LIN {X 0,Y 333.716,Z 810.919,A -85,B 0,C 180,E1 -14697.808,E2 -14697.808} C_VEL
LIN {X 0,Y 333.692,Z 810.92,A -85,B 0,C 180,E1 -14700.36,E2 -14700.36} C_VEL
LIN {X 0,Y 333.667,Z 810.922,A -85,B 0,C 180,E1 -14704.656,E2 -14704.656} C_VEL
LIN {X 0,Y 333.648,Z 810.925,A -85,B 0,C 180,E1 -14707.648,E2 -14707.648} C_VEL
LIN {X 0,Y 333.69,Z 810.919,A -85,B 0,C 180,E1 -14710.757,E2 -14710.757} C_VEL
LIN {X 0,Y 333.72,Z 810.918,A -85,B 0,C 180,E1 -14714.272,E2 -14714.272} C_VEL
LIN {X 0,Y 333.695,Z 810.911,A -85,B 0,C 180,E1 -14717.627,E2 -14717.627} C_VEL
LIN {X 0,Y 333.676,Z 810.914,A -85,B 0,C 180,E1 -14721.193,E2 -14721.193} C_VEL
LIN {X 0,Y 333.644,Z 810.921,A -85,B 0,C 180,E1 -14722.65,E2 -14722.65} C_VEL
LIN {X 0,Y 332.983,Z 811.005,A -85,B 0,C 180,E1 -14723.657,E2 -14723.657} C_VEL
LIN {X 0,Y 330.131,Z 811.362,A -85,B 0,C 180,E1 -14725.297,E2 -14725.297} C_VEL
LIN {X 0,Y 327.705,Z 811.662,A -85,B 0,C 180,E1 -14726.625,E2 -14726.625} C_VEL
LIN {X 0,Y 326.655,Z 811.793,A -85,B 0,C 180,E1 -14727.654,E2 -14727.654} C_VEL
LIN {X 0,Y 326.565,Z 811.801,A -85,B 0,C 180,E1 -14728.002,E2 -14728.002} C_VEL
LIN {X 0,Y 326.643,Z 811.794,A -85,B 0,C 180,E1 -14731.748,E2 -14731.748} C_VEL
LIN {X 0,Y 326.674,Z 811.789,A -85,B 0,C 180,E1 -14734.626,E2 -14734.626} C_VEL
LIN {X 0,Y 326.633,Z 811.797,A -85,B 0,C 180,E1 -14738.544,E2 -14738.544} C_VEL
LIN {X 0,Y 326.729,Z 811.788,A -85,B 0,C 180,E1 -14741.176,E2 -14741.176} C_VEL
LIN {X 0,Y 326.747,Z 811.778,A -85,B 0,C 180,E1 -14745.432,E2 -14745.432} C_VEL
LIN {X 0,Y 326.758,Z 811.784,A -85,B 0,C 180,E1 -14748.838,E2 -14748.838} C_VEL
LIN {X 0,Y 326.949,Z 811.757,A -85,B 0,C 180,E1 -14752.59,E2 -14752.59} C_VEL
LIN {X 0,Y 326.76,Z 811.787,A -85,B 0,C 180,E1 -14755.065,E2 -14755.065} C_VEL
LIN {X 0,Y 327.03,Z 811.746,A -85,B 0,C 180,E1 -14757.537,E2 -14757.537} C_VEL
LIN {X 0,Y 327.181,Z 811.733,A -85,B 0,C 180,E1 -14760,E2 -14760} C_VEL
LIN {X 0,Y 327.029,Z 811.75,A -85,B 0,C 180,E1 -14762.463,E2 -14762.463} C_VEL
LIN {X 0,Y 326.945,Z 811.758,A -85,B 0,C 180,E1 -14766.17,E2 -14766.17} C_VEL
LIN {X 0,Y 326.898,Z 811.762,A -85,B 0,C 180,E1 -14768.655,E2 -14768.655} C_VEL
LIN {X 0,Y 326.721,Z 811.78,A -85,B 0,C 180,E1 -14772.422,E2 -14772.422} C_VEL
LIN {X 0,Y 326.738,Z 811.784,A -85,B 0,C 180,E1 -14774.958,E2 -14774.958} C_VEL
LIN {X 0,Y 326.717,Z 811.788,A -85,B 0,C 180,E1 -14778.839,E2 -14778.839} C_VEL
LIN {X 0,Y 326.582,Z 811.804,A -85,B 0,C 180,E1 -14782.79,E2 -14782.79} C_VEL
LIN {X 0,Y 326.619,Z 811.798,A -85,B 0,C 180,E1 -14785.49,E2 -14785.49} C_VEL
LIN {X 0,Y 326.601,Z 811.803,A -85,B 0,C 180,E1 -14789.665,E2 -14789.665} C_VEL
LIN {X 0,Y 326.603,Z 811.8,A -85,B 0,C 180,E1 -14792.947,E2 -14792.947} C_VEL
LIN {X 0,Y 326.596,Z 811.803,A -85,B 0,C 180,E1 -14795.522,E2 -14795.522} C_VEL
LIN {X 0,Y 326.573,Z 811.807,A -85,B 0,C 180,E1 -14799.223,E2 -14799.223} C_VEL
LIN {X 0,Y 326.595,Z 811.905,A -85,B 0,C 180,E1 -14801.33,E2 -14801.33} C_VEL
LIN {X 0,Y 327.886,Z 817.95,A -85,B 0,C 180,E1 -14804.156,E2 -14804.156} C_VEL
LIN {X 0,Y 329.434,Z 825.489,A -85,B 0,C 180,E1 -14807.477,E2 -14807.477} C_VEL
LIN {X 0,Y 331.048,Z 834.395,A -85,B 0,C 180,E1 -14811.14,E2 -14811.14} C_VEL
LIN {X 0,Y 331.312,Z 837.705,A -85,B 0,C 180,E1 -14812.424,E2 -14812.424} C_VEL
LIN {X 0,Y 329.861,Z 848.572,A -85,B 0,C 180,E1 -14816.364,E2 -14816.364} C_VEL
LIN {X 0,Y 328.321,Z 861.677,A -85,B 0,C 180,E1 -14821.019,E2 -14821.019} C_VEL
LIN {X 0,Y 327.361,Z 871.737,A -85,B 0,C 180,E1 -14824.575,E2 -14824.575} C_VEL
LIN {X 0,Y 326.643,Z 880.438,A -85,B 0,C 180,E1 -14827.625,E2 -14827.625} C_VEL
LIN {X 0,Y 328.711,Z 894.714,A -85,B 0,C 180,E1 -14828.278,E2 -14828.278} C_VEL
LIN {X 0,Y 329.806,Z 906.751,A -85,B 0,C 180,E1 -14829.017,E2 -14829.017} C_VEL
LIN {X 0,Y 330.337,Z 918.761,A -85,B 0,C 180,E1 -14829.954,E2 -14829.954} C_VEL
LIN {X 0,Y 330.378,Z 930.265,A -85,B 0,C 180,E1 -14831.073,E2 -14831.073} C_VEL
LIN {X 0,Y 330.455,Z 937.231,A -85,B 0,C 180,E1 -14831.881,E2 -14831.881} C_VEL
LIN {X 0,Y 329.062,Z 947.55,A -85,B 0,C 180,E1 -14833.245,E2 -14833.245} C_VEL
LIN {X 0,Y 327.748,Z 957.445,A -85,B 0,C 180,E1 -14834.881,E2 -14834.881} C_VEL
LIN {X 0,Y 326.998,Z 964.642,A -85,B 0,C 180,E1 -14836.327,E2 -14836.327} C_VEL
LIN {X 0,Y 326.251,Z 972.29,A -85,B 0,C 180,E1 -14838.194,E2 -14838.194} C_VEL
LIN {X 0,Y 325.834,Z 978.472,A -85,B 0,C 180,E1 -14840.066,E2 -14840.066} C_VEL
LIN {X 0,Y 325.696,Z 983.394,A -85,B 0,C 180,E1 -14841.939,E2 -14841.939} C_VEL
LIN {X 0,Y 325.738,Z 987.186,A -85,B 0,C 180,E1 -14843.809,E2 -14843.809} C_VEL
LIN {X 0,Y 325.892,Z 989.16,A -85,B 0,C 180,E1 -14845.054,E2 -14845.054} C_VEL
LIN {X 0,Y 326.004,Z 990.64,A -85,B 0,C 180,E1 -14846.294,E2 -14846.294} C_VEL
LIN {X 0,Y 326.056,Z 991.691,A -85,B 0,C 180,E1 -14847.532,E2 -14847.532} C_VEL
LIN {X 0,Y 326.14,Z 992.338,A -85,B 0,C 180,E1 -14848.767,E2 -14848.767} C_VEL
LIN {X 0,Y 326.213,Z 992.572,A -85,B 0,C 180,E1 -14850.002,E2 -14850.002} C_VEL
LIN {X 0,Y 326.141,Z 992.332,A -85,B 0,C 180,E1 -14851.237,E2 -14851.237} C_VEL
LIN {X 0,Y 326.057,Z 991.679,A -85,B 0,C 180,E1 -14852.473,E2 -14852.473} C_VEL
LIN {X 0,Y 326.005,Z 990.623,A -85,B 0,C 180,E1 -14853.71,E2 -14853.71} C_VEL
LIN {X 0,Y 325.893,Z 989.136,A -85,B 0,C 180,E1 -14854.951,E2 -14854.951} C_VEL
LIN {X 0,Y 325.738,Z 985.606,A -85,B 0,C 180,E1 -14857.03,E2 -14857.03} C_VEL
LIN {X 0,Y 325.757,Z 980.196,A -85,B 0,C 180,E1 -14859.314,E2 -14859.314} C_VEL
LIN {X 0,Y 326.028,Z 974.442,A -85,B 0,C 180,E1 -14861.189,E2 -14861.189} C_VEL
LIN {X 0,Y 326.71,Z 967.329,A -85,B 0,C 180,E1 -14863.056,E2 -14863.056} C_VEL
LIN {X 0,Y 327.555,Z 960.109,A -85,B 0,C 180,E1 -14864.604,E2 -14864.604} C_VEL
LIN {X 0,Y 329.351,Z 946.504,A -85,B 0,C 180,E1 -14867.064,E2 -14867.064} C_VEL
LIN {X 0,Y 330.884,Z 936.373,A -85,B 0,C 180,E1 -14868.58,E2 -14868.58} C_VEL
LIN {X 0,Y 331.378,Z 923.905,A -85,B 0,C 180,E1 -14870.201,E2 -14870.201} C_VEL
LIN {X 0,Y 331.81,Z 912.737,A -85,B 0,C 180,E1 -14871.432,E2 -14871.432} C_VEL
LIN {X 0,Y 331.901,Z 904.635,A -85,B 0,C 180,E1 -14872.243,E2 -14872.243} C_VEL
LIN {X 0,Y 330.655,Z 891.44,A -85,B 0,C 180,E1 -14873.499,E2 -14873.499} C_VEL
LIN {X 0,Y 328.27,Z 877.306,A -85,B 0,C 180,E1 -14874.788,E2 -14874.788} C_VEL
LIN {X 0,Y 327.341,Z 873.127,A -85,B 0,C 180,E1 -14875.176,E2 -14875.176} C_VEL
LIN {X 0,Y 327.288,Z 872.165,A -85,B 0,C 180,E1 -14875.266,E2 -14875.266} C_VEL
LIN {X 0,Y 328.289,Z 861.638,A -85,B 0,C 180,E1 -14878.985,E2 -14878.985} C_VEL
LIN {X 0,Y 329.588,Z 850.492,A -85,B 0,C 180,E1 -14882.941,E2 -14882.941} C_VEL
LIN {X 0,Y 331.19,Z 838.637,A -85,B 0,C 180,E1 -14887.215,E2 -14887.215} C_VEL
LIN {X 0,Y 331.22,Z 835.828,A -85,B 0,C 180,E1 -14888.271,E2 -14888.271} C_VEL
LIN {X 0,Y 329.746,Z 827.239,A -85,B 0,C 180,E1 -14891.758,E2 -14891.758} C_VEL
LIN {X 0,Y 327.846,Z 817.89,A -85,B 0,C 180,E1 -14895.837,E2 -14895.837} C_VEL
LIN {X 0,Y 326.561,Z 811.81,A -85,B 0,C 180,E1 -14898.772,E2 -14898.772} C_VEL
LIN {X 0,Y 326.629,Z 811.798,A -85,B 0,C 180,E1 -14902.953,E2 -14902.953} C_VEL
LIN {X 0,Y 326.611,Z 811.799,A -85,B 0,C 180,E1 -14905.981,E2 -14905.981} C_VEL
LIN {X 0,Y 326.616,Z 811.799,A -85,B 0,C 180,E1 -14909.399,E2 -14909.399} C_VEL
LIN {X 0,Y 326.6,Z 811.803,A -85,B 0,C 180,E1 -14913.135,E2 -14913.135} C_VEL
LIN {X 0,Y 326.614,Z 811.858,A -85,B 0,C 180,E1 -14914.424,E2 -14914.424} C_VEL
LIN {X 0,Y 326.863,Z 813.01,A -85,B 0,C 180,E1 -14914.566,E2 -14914.566} C_VEL
LIN {X 0,Y 327.872,Z 815.002,A -85,B 0,C 180,E1 -14914.913,E2 -14914.913} C_VEL
LIN {X 0,Y 329.004,Z 816.271,A -85,B 0,C 180,E1 -14915.215,E2 -14915.215} C_VEL
LIN {X 0,Y 331.968,Z 822.323,A -85,B 0,C 180,E1 -14916.281,E2 -14916.281} C_VEL
LIN {X 0,Y 335.858,Z 830.631,A -85,B 0,C 180,E1 -14917.76,E2 -14917.76} C_VEL
LIN {X 0,Y 339.022,Z 840.104,A -85,B 0,C 180,E1 -14919.365,E2 -14919.365} C_VEL
LIN {X 0,Y 339.722,Z 843.27,A -85,B 0,C 180,E1 -14919.896,E2 -14919.896} C_VEL
LIN {X 0,Y 338.28,Z 853.109,A -85,B 0,C 180,E1 -14921.215,E2 -14921.215} C_VEL
LIN {X 0,Y 336.922,Z 860.61,A -85,B 0,C 180,E1 -14922.394,E2 -14922.394} C_VEL
LIN {X 0,Y 335.4,Z 868.603,A -85,B 0,C 180,E1 -14923.88,E2 -14923.88} C_VEL
LIN {X 0,Y 333.761,Z 876.022,A -85,B 0,C 180,E1 -14925.614,E2 -14925.614} C_VEL
LIN {X 0,Y 332.03,Z 883.463,A -85,B 0,C 180,E1 -14927.78,E2 -14927.78} C_VEL
LIN {X 0,Y 330.34,Z 889.554,A -85,B 0,C 180,E1 -14930.201,E2 -14930.201} C_VEL
LIN {X 0,Y 329.629,Z 891.806,A -85,B 0,C 180,E1 -14931.417,E2 -14931.417} C_VEL
LIN {X 0,Y 328.897,Z 893.676,A -85,B 0,C 180,E1 -14932.634,E2 -14932.634} C_VEL
LIN {X 0,Y 328.111,Z 896.009,A -85,B 0,C 180,E1 -14935.085,E2 -14935.085} C_VEL
LIN {X 0,Y 327.478,Z 896.771,A -85,B 0,C 180,E1 -14937.54,E2 -14937.54} C_VEL
LIN {X 0,Y 327.203,Z 896.509,A -85,B 0,C 180,E1 -14938.769,E2 -14938.769} C_VEL
LIN {X 0,Y 326.915,Z 895.854,A -85,B 0,C 180,E1 -14940,E2 -14940} C_VEL
LIN {X 0,Y 326.782,Z 893.268,A -85,B 0,C 180,E1 -14942.465,E2 -14942.465} C_VEL
LIN {X 0,Y 326.755,Z 890.202,A -85,B 0,C 180,E1 -14944.317,E2 -14944.317} C_VEL
LIN {X 0,Y 327.16,Z 886.056,A -85,B 0,C 180,E1 -14946.166,E2 -14946.166} C_VEL
LIN {X 0,Y 327.526,Z 880.773,A -85,B 0,C 180,E1 -14948.018,E2 -14948.018} C_VEL
LIN {X 0,Y 327.848,Z 875.453,A -85,B 0,C 180,E1 -14949.559,E2 -14949.559} C_VEL
LIN {X 0,Y 328.493,Z 867.671,A -85,B 0,C 180,E1 -14951.414,E2 -14951.414} C_VEL
LIN {X 0,Y 329.086,Z 859.694,A -85,B 0,C 180,E1 -14952.958,E2 -14952.958} C_VEL
LIN {X 0,Y 329.713,Z 851.26,A -85,B 0,C 180,E1 -14954.347,E2 -14954.347} C_VEL
LIN {X 0,Y 330.285,Z 843.596,A -85,B 0,C 180,E1 -14955.425,E2 -14955.425} C_VEL
LIN {X 0,Y 331.05,Z 833.535,A -85,B 0,C 180,E1 -14956.638,E2 -14956.638} C_VEL
LIN {X 0,Y 331.244,Z 830.494,A -85,B 0,C 180,E1 -14956.954,E2 -14956.954} C_VEL
LIN {X 0,Y 328.32,Z 818.286,A -85,B 0,C 180,E1 -14958.217,E2 -14958.217} C_VEL
LIN {X 0,Y 326.633,Z 811.795,A -85,B 0,C 180,E1 -14958.806,E2 -14958.806} C_VEL
LIN {X 0,Y 326.59,Z 811.797,A -85,B 0,C 180,E1 -14962.79,E2 -14962.79} C_VEL
LIN {X 0,Y 326.601,Z 811.792,A -85,B 0,C 180,E1 -14966.865,E2 -14966.865} C_VEL
LIN {X 0,Y 326.58,Z 811.8,A -85,B 0,C 180,E1 -14971.097,E2 -14971.097} C_VEL
LIN {X 0,Y 326.613,Z 811.796,A -85,B 0,C 180,E1 -14974.019,E2 -14974.019} C_VEL
LIN {X 0,Y 326.628,Z 811.791,A -85,B 0,C 180,E1 -14977.236,E2 -14977.236} C_VEL
LIN {X 0,Y 326.551,Z 811.804,A -85,B 0,C 180,E1 -14981.124,E2 -14981.124} C_VEL
LIN {X 0,Y 326.568,Z 811.802,A -85,B 0,C 180,E1 -14983.525,E2 -14983.525} C_VEL
LIN {X 0,Y 326.581,Z 811.801,A -85,B 0,C 180,E1 -14987.028,E2 -14987.028} C_VEL
LIN {X 0,Y 326.593,Z 811.802,A -85,B 0,C 180,E1 -14990.777,E2 -14990.777} C_VEL
LIN {X 0,Y 326.619,Z 811.801,A -85,B 0,C 180,E1 -14994.479,E2 -14994.479} C_VEL
LIN {X 0,Y 326.615,Z 811.797,A -85,B 0,C 180,E1 -14997.454,E2 -14997.454} C_VEL
LIN {X 0,Y 326.654,Z 811.79,A -85,B 0,C 180,E1 -15000.338,E2 -15000.338} C_VEL
LIN {X 0,Y 326.696,Z 811.783,A -85,B 0,C 180,E1 -15004.515,E2 -15004.515} C_VEL
LIN {X 0,Y 326.65,Z 811.826,A -85,B 0,C 180,E1 -15008.544,E2 -15008.544} C_VEL
LIN {X 0,Y 330.897,Z 823.77,A -85,B 0,C 180,E1 -15009.727,E2 -15009.727} C_VEL
LIN {X 0,Y 334.128,Z 834.117,A -85,B 0,C 180,E1 -15010.94,E2 -15010.94} C_VEL
LIN {X 0,Y 334.837,Z 836.764,A -85,B 0,C 180,E1 -15011.276,E2 -15011.276} C_VEL
LIN {X 0,Y 333.841,Z 847.507,A -85,B 0,C 180,E1 -15012.541,E2 -15012.541} C_VEL
LIN {X 0,Y 332.661,Z 857.844,A -85,B 0,C 180,E1 -15014.057,E2 -15014.057} C_VEL
LIN {X 0,Y 331.579,Z 866.207,A -85,B 0,C 180,E1 -15015.577,E2 -15015.577} C_VEL
LIN {X 0,Y 330.347,Z 874.325,A -85,B 0,C 180,E1 -15017.403,E2 -15017.403} C_VEL
LIN {X 0,Y 329.595,Z 879.852,A -85,B 0,C 180,E1 -15018.934,E2 -15018.934} C_VEL
LIN {X 0,Y 328.829,Z 885.233,A -85,B 0,C 180,E1 -15020.774,E2 -15020.774} C_VEL
LIN {X 0,Y 327.901,Z 889.497,A -85,B 0,C 180,E1 -15022.609,E2 -15022.609} C_VEL
LIN {X 0,Y 327.572,Z 891.723,A -85,B 0,C 180,E1 -15023.84,E2 -15023.84} C_VEL
LIN {X 0,Y 327.275,Z 893.539,A -85,B 0,C 180,E1 -15025.07,E2 -15025.07} C_VEL
LIN {X 0,Y 327.271,Z 894.875,A -85,B 0,C 180,E1 -15026.304,E2 -15026.304} C_VEL
LIN {X 0,Y 326.973,Z 896.453,A -85,B 0,C 180,E1 -15028.766,E2 -15028.766} C_VEL
LIN {X 0,Y 326.926,Z 896.684,A -85,B 0,C 180,E1 -15029.998,E2 -15029.998} C_VEL
LIN {X 0,Y 327.106,Z 895.92,A -85,B 0,C 180,E1 -15032.461,E2 -15032.461} C_VEL
LIN {X 0,Y 327.23,Z 894.981,A -85,B 0,C 180,E1 -15033.692,E2 -15033.692} C_VEL
LIN {X 0,Y 327.263,Z 893.685,A -85,B 0,C 180,E1 -15034.926,E2 -15034.926} C_VEL
LIN {X 0,Y 327.73,Z 890.88,A -85,B 0,C 180,E1 -15036.771,E2 -15036.771} C_VEL
LIN {X 0,Y 328.576,Z 887.039,A -85,B 0,C 180,E1 -15038.609,E2 -15038.609} C_VEL
LIN {X 0,Y 329.297,Z 882.586,A -85,B 0,C 180,E1 -15040.287,E2 -15040.287} C_VEL
LIN {X 0,Y 330.101,Z 875.962,A -85,B 0,C 180,E1 -15042.29,E2 -15042.29} C_VEL
LIN {X 0,Y 331.295,Z 868.186,A -85,B 0,C 180,E1 -15044.118,E2 -15044.118} C_VEL
LIN {X 0,Y 332.365,Z 860.257,A -85,B 0,C 180,E1 -15045.638,E2 -15045.638} C_VEL
LIN {X 0,Y 333.544,Z 850.564,A -85,B 0,C 180,E1 -15047.154,E2 -15047.154} C_VEL
LIN {X 0,Y 334.7,Z 839.753,A -85,B 0,C 180,E1 -15048.501,E2 -15048.501} C_VEL
LIN {X 0,Y 334.99,Z 837.259,A -85,B 0,C 180,E1 -15048.765,E2 -15048.765} C_VEL
LIN {X 0,Y 331.653,Z 825.781,A -85,B 0,C 180,E1 -15050.157,E2 -15050.157} C_VEL
LIN {X 0,Y 327.543,Z 814.401,A -85,B 0,C 180,E1 -15051.331,E2 -15051.331} C_VEL
LIN {X 0,Y 326.666,Z 811.794,A -85,B 0,C 180,E1 -15051.573,E2 -15051.573} C_VEL
LIN {X 0,Y 326.686,Z 811.793,A -85,B 0,C 180,E1 -15055.481,E2 -15055.481} C_VEL
LIN {X 0,Y 326.655,Z 811.797,A -85,B 0,C 180,E1 -15059.657,E2 -15059.657} C_VEL
LIN {X 0,Y 326.601,Z 811.805,A -85,B 0,C 180,E1 -15064.017,E2 -15064.017} C_VEL
LIN {X 0,Y 326.622,Z 811.799,A -85,B 0,C 180,E1 -15067.237,E2 -15067.237} C_VEL
LIN {X 0,Y 326.627,Z 811.802,A -85,B 0,C 180,E1 -15070.2,E2 -15070.2} C_VEL
LIN {X 0,Y 326.649,Z 811.795,A -85,B 0,C 180,E1 -15073.507,E2 -15073.507} C_VEL
LIN {X 0,Y 326.64,Z 811.791,A -85,B 0,C 180,E1 -15077.012,E2 -15077.012} C_VEL
LIN {X 0,Y 326.636,Z 811.793,A -85,B 0,C 180,E1 -15080.763,E2 -15080.763} C_VEL
LIN {X 0,Y 326.602,Z 811.801,A -85,B 0,C 180,E1 -15084.479,E2 -15084.479} C_VEL
LIN {X 0,Y 326.565,Z 811.801,A -85,B 0,C 180,E1 -15088.002,E2 -15088.002} C_VEL
LIN {X 0,Y 325.885,Z 811.888,A -85,B 0,C 180,E1 -15089.033,E2 -15089.033} C_VEL
LIN {X 0,Y 323.038,Z 812.242,A -85,B 0,C 180,E1 -15090.711,E2 -15090.711} C_VEL
LIN {X 0,Y 320.653,Z 812.541,A -85,B 0,C 180,E1 -15092.07,E2 -15092.07} C_VEL
LIN {X 0,Y 319.658,Z 812.664,A -85,B 0,C 180,E1 -15093.122,E2 -15093.122} C_VEL
LIN {X 0,Y 319.592,Z 812.669,A -85,B 0,C 180,E1 -15093.478,E2 -15093.478} C_VEL
LIN {X 0,Y 319.594,Z 812.673,A -85,B 0,C 180,E1 -15097.45,E2 -15097.45} C_VEL
LIN {X 0,Y 319.674,Z 812.665,A -85,B 0,C 180,E1 -15100.961,E2 -15100.961} C_VEL
LIN {X 0,Y 319.715,Z 812.653,A -85,B 0,C 180,E1 -15105.275,E2 -15105.275} C_VEL
LIN {X 0,Y 319.743,Z 812.65,A -85,B 0,C 180,E1 -15109.872,E2 -15109.872} C_VEL
LIN {X 0,Y 319.908,Z 812.634,A -85,B 0,C 180,E1 -15112.426,E2 -15112.426} C_VEL
LIN {X 0,Y 319.729,Z 812.662,A -85,B 0,C 180,E1 -15114.956,E2 -15114.956} C_VEL
LIN {X 0,Y 319.974,Z 812.625,A -85,B 0,C 180,E1 -15117.482,E2 -15117.482} C_VEL
LIN {X 0,Y 320.133,Z 812.611,A -85,B 0,C 180,E1 -15120,E2 -15120} C_VEL
LIN {X 0,Y 319.972,Z 812.629,A -85,B 0,C 180,E1 -15122.518,E2 -15122.518} C_VEL
LIN {X 0,Y 319.905,Z 812.634,A -85,B 0,C 180,E1 -15126.306,E2 -15126.306} C_VEL
LIN {X 0,Y 319.826,Z 812.644,A -85,B 0,C 180,E1 -15128.848,E2 -15128.848} C_VEL
LIN {X 0,Y 319.668,Z 812.658,A -85,B 0,C 180,E1 -15132.7,E2 -15132.7} C_VEL
LIN {X 0,Y 319.683,Z 812.664,A -85,B 0,C 180,E1 -15135.296,E2 -15135.296} C_VEL
LIN {X 0,Y 319.636,Z 812.671,A -85,B 0,C 180,E1 -15139.257,E2 -15139.257} C_VEL
LIN {X 0,Y 319.535,Z 812.682,A -85,B 0,C 180,E1 -15143.322,E2 -15143.322} C_VEL
LIN {X 0,Y 319.555,Z 812.682,A -85,B 0,C 180,E1 -15146.095,E2 -15146.095} C_VEL
LIN {X 0,Y 319.528,Z 812.683,A -85,B 0,C 180,E1 -15148.94,E2 -15148.94} C_VEL
LIN {X 0,Y 319.51,Z 812.687,A -85,B 0,C 180,E1 -15151.864,E2 -15151.864} C_VEL
LIN {X 0,Y 319.564,Z 812.679,A -85,B 0,C 180,E1 -15155.544,E2 -15155.544} C_VEL
LIN {X 0,Y 319.515,Z 812.685,A -85,B 0,C 180,E1 -15159.664,E2 -15159.664} C_VEL
LIN {X 0,Y 319.516,Z 812.77,A -85,B 0,C 180,E1 -15160.768,E2 -15160.768} C_VEL
LIN {X 0,Y 320.852,Z 818.876,A -85,B 0,C 180,E1 -15163.715,E2 -15163.715} C_VEL
LIN {X 0,Y 322.555,Z 827.284,A -85,B 0,C 180,E1 -15167.515,E2 -15167.515} C_VEL
LIN {X 0,Y 324.156,Z 836.315,A -85,B 0,C 180,E1 -15171.308,E2 -15171.308} C_VEL
LIN {X 0,Y 324.37,Z 838.045,A -85,B 0,C 180,E1 -15171.999,E2 -15171.999} C_VEL
LIN {X 0,Y 323.005,Z 848.16,A -85,B 0,C 180,E1 -15175.773,E2 -15175.773} C_VEL
LIN {X 0,Y 321.411,Z 861.126,A -85,B 0,C 180,E1 -15180.51,E2 -15180.51} C_VEL
LIN {X 0,Y 320.381,Z 870.951,A -85,B 0,C 180,E1 -15184.078,E2 -15184.078} C_VEL
LIN {X 0,Y 319.658,Z 879.219,A -85,B 0,C 180,E1 -15187.102,E2 -15187.102} C_VEL
LIN {X 0,Y 321.715,Z 893.437,A -85,B 0,C 180,E1 -15187.773,E2 -15187.773} C_VEL
LIN {X 0,Y 322.964,Z 906.575,A -85,B 0,C 180,E1 -15188.611,E2 -15188.611} C_VEL
LIN {X 0,Y 323.473,Z 919.342,A -85,B 0,C 180,E1 -15189.66,E2 -15189.66} C_VEL
LIN {X 0,Y 323.455,Z 932.128,A -85,B 0,C 180,E1 -15190.981,E2 -15190.981} C_VEL
LIN {X 0,Y 323.493,Z 937.462,A -85,B 0,C 180,E1 -15191.641,E2 -15191.641} C_VEL
LIN {X 0,Y 321.942,Z 948.492,A -85,B 0,C 180,E1 -15193.19,E2 -15193.19} C_VEL
LIN {X 0,Y 320.675,Z 957.492,A -85,B 0,C 180,E1 -15194.755,E2 -15194.755} C_VEL
LIN {X 0,Y 319.852,Z 964.981,A -85,B 0,C 180,E1 -15196.34,E2 -15196.34} C_VEL
LIN {X 0,Y 319.135,Z 972.391,A -85,B 0,C 180,E1 -15198.249,E2 -15198.249} C_VEL
LIN {X 0,Y 318.703,Z 979.188,A -85,B 0,C 180,E1 -15200.483,E2 -15200.483} C_VEL
LIN {X 0,Y 318.624,Z 983.725,A -85,B 0,C 180,E1 -15202.397,E2 -15202.397} C_VEL
LIN {X 0,Y 318.678,Z 986.144,A -85,B 0,C 180,E1 -15203.672,E2 -15203.672} C_VEL
LIN {X 0,Y 318.84,Z 988.121,A -85,B 0,C 180,E1 -15204.944,E2 -15204.944} C_VEL
LIN {X 0,Y 318.962,Z 989.604,A -85,B 0,C 180,E1 -15206.212,E2 -15206.212} C_VEL
LIN {X 0,Y 319.015,Z 990.656,A -85,B 0,C 180,E1 -15207.477,E2 -15207.477} C_VEL
LIN {X 0,Y 319.107,Z 991.305,A -85,B 0,C 180,E1 -15208.74,E2 -15208.74} C_VEL
LIN {X 0,Y 319.187,Z 991.541,A -85,B 0,C 180,E1 -15210.002,E2 -15210.002} C_VEL
LIN {X 0,Y 319.107,Z 991.299,A -85,B 0,C 180,E1 -15211.264,E2 -15211.264} C_VEL
LIN {X 0,Y 319.016,Z 990.644,A -85,B 0,C 180,E1 -15212.528,E2 -15212.528} C_VEL
LIN {X 0,Y 318.963,Z 989.587,A -85,B 0,C 180,E1 -15213.792,E2 -15213.792} C_VEL
LIN {X 0,Y 318.841,Z 988.096,A -85,B 0,C 180,E1 -15215.06,E2 -15215.06} C_VEL
LIN {X 0,Y 318.683,Z 984.801,A -85,B 0,C 180,E1 -15217.068,E2 -15217.068} C_VEL
LIN {X 0,Y 318.649,Z 980.811,A -85,B 0,C 180,E1 -15218.884,E2 -15218.884} C_VEL
LIN {X 0,Y 318.933,Z 974.437,A -85,B 0,C 180,E1 -15221.119,E2 -15221.119} C_VEL
LIN {X 0,Y 319.599,Z 967.549,A -85,B 0,C 180,E1 -15223.028,E2 -15223.028} C_VEL
LIN {X 0,Y 321.045,Z 956.136,A -85,B 0,C 180,E1 -15225.591,E2 -15225.591} C_VEL
LIN {X 0,Y 322.246,Z 948.288,A -85,B 0,C 180,E1 -15227.125,E2 -15227.125} C_VEL
LIN {X 0,Y 324.034,Z 937.615,A -85,B 0,C 180,E1 -15228.824,E2 -15228.824} C_VEL
LIN {X 0,Y 324.586,Z 927.478,A -85,B 0,C 180,E1 -15230.271,E2 -15230.271} C_VEL
LIN {X 0,Y 325.373,Z 914.236,A -85,B 0,C 180,E1 -15231.877,E2 -15231.877} C_VEL
LIN {X 0,Y 325.477,Z 903.651,A -85,B 0,C 180,E1 -15232.999,E2 -15232.999} C_VEL
LIN {X 0,Y 324.001,Z 888.952,A -85,B 0,C 180,E1 -15234.494,E2 -15234.494} C_VEL
LIN {X 0,Y 322.117,Z 878.146,A -85,B 0,C 180,E1 -15235.587,E2 -15235.587} C_VEL
LIN {X 0,Y 321.217,Z 873.894,A -85,B 0,C 180,E1 -15236.005,E2 -15236.005} C_VEL
LIN {X 0,Y 320.491,Z 869.527,A -85,B 0,C 180,E1 -15236.426,E2 -15236.426} C_VEL
LIN {X 0,Y 321.344,Z 861.087,A -85,B 0,C 180,E1 -15239.496,E2 -15239.496} C_VEL
LIN {X 0,Y 322.79,Z 849.786,A -85,B 0,C 180,E1 -15243.614,E2 -15243.614} C_VEL
LIN {X 0,Y 324.218,Z 839.641,A -85,B 0,C 180,E1 -15247.371,E2 -15247.371} C_VEL
LIN {X 0,Y 324.144,Z 836.27,A -85,B 0,C 180,E1 -15248.69,E2 -15248.69} C_VEL
LIN {X 0,Y 322.631,Z 827.856,A -85,B 0,C 180,E1 -15252.214,E2 -15252.214} C_VEL
LIN {X 0,Y 320.778,Z 818.703,A -85,B 0,C 180,E1 -15256.305,E2 -15256.305} C_VEL
LIN {X 0,Y 319.497,Z 812.687,A -85,B 0,C 180,E1 -15259.333,E2 -15259.333} C_VEL
LIN {X 0,Y 319.56,Z 812.676,A -85,B 0,C 180,E1 -15263.572,E2 -15263.572} C_VEL
LIN {X 0,Y 319.584,Z 812.679,A -85,B 0,C 180,E1 -15266.688,E2 -15266.688} C_VEL
LIN {X 0,Y 319.557,Z 812.678,A -85,B 0,C 180,E1 -15269.613,E2 -15269.613} C_VEL
LIN {X 0,Y 319.563,Z 812.731,A -85,B 0,C 180,E1 -15273.07,E2 -15273.07} C_VEL
LIN {X 0,Y 320.392,Z 815.235,A -85,B 0,C 180,E1 -15273.477,E2 -15273.477} C_VEL
LIN {X 0,Y 322.496,Z 818.125,A -85,B 0,C 180,E1 -15274.161,E2 -15274.161} C_VEL
LIN {X 0,Y 323.497,Z 820.131,A -85,B 0,C 180,E1 -15274.532,E2 -15274.532} C_VEL
LIN {X 0,Y 324.412,Z 821.332,A -85,B 0,C 180,E1 -15274.836,E2 -15274.836} C_VEL
LIN {X 0,Y 329.008,Z 831.134,A -85,B 0,C 180,E1 -15276.716,E2 -15276.716} C_VEL
LIN {X 0,Y 331.671,Z 838.229,A -85,B 0,C 180,E1 -15278.024,E2 -15278.024} C_VEL
LIN {X 0,Y 333.604,Z 845.299,A -85,B 0,C 180,E1 -15279.302,E2 -15279.302} C_VEL
LIN {X 0,Y 333.404,Z 848.069,A -85,B 0,C 180,E1 -15279.696,E2 -15279.696} C_VEL
LIN {X 0,Y 331.63,Z 858.133,A -85,B 0,C 180,E1 -15281.144,E2 -15281.144} C_VEL
LIN {X 0,Y 329.59,Z 868.152,A -85,B 0,C 180,E1 -15282.95,E2 -15282.95} C_VEL
LIN {X 0,Y 327.921,Z 875.173,A -85,B 0,C 180,E1 -15284.524,E2 -15284.524} C_VEL
LIN {X 0,Y 326.354,Z 881.609,A -85,B 0,C 180,E1 -15286.297,E2 -15286.297} C_VEL
LIN {X 0,Y 324.878,Z 886.983,A -85,B 0,C 180,E1 -15288.141,E2 -15288.141} C_VEL
LIN {X 0,Y 323.565,Z 891.28,A -85,B 0,C 180,E1 -15289.993,E2 -15289.993} C_VEL
LIN {X 0,Y 322.055,Z 895.256,A -85,B 0,C 180,E1 -15292.476,E2 -15292.476} C_VEL
LIN {X 0,Y 321.19,Z 897.358,A -85,B 0,C 180,E1 -15294.979,E2 -15294.979} C_VEL
LIN {X 0,Y 320.839,Z 897.896,A -85,B 0,C 180,E1 -15296.232,E2 -15296.232} C_VEL
LIN {X 0,Y 320.492,Z 897.979,A -85,B 0,C 180,E1 -15297.486,E2 -15297.486} C_VEL
LIN {X 0,Y 320.213,Z 897.636,A -85,B 0,C 180,E1 -15298.742,E2 -15298.742} C_VEL
LIN {X 0,Y 319.896,Z 896.917,A -85,B 0,C 180,E1 -15300,E2 -15300} C_VEL
LIN {X 0,Y 319.757,Z 894.125,A -85,B 0,C 180,E1 -15302.52,E2 -15302.52} C_VEL
LIN {X 0,Y 319.736,Z 890.932,A -85,B 0,C 180,E1 -15304.412,E2 -15304.412} C_VEL
LIN {X 0,Y 320.126,Z 886.656,A -85,B 0,C 180,E1 -15306.302,E2 -15306.302} C_VEL
LIN {X 0,Y 320.512,Z 881.235,A -85,B 0,C 180,E1 -15308.194,E2 -15308.194} C_VEL
LIN {X 0,Y 320.813,Z 876.216,A -85,B 0,C 180,E1 -15309.656,E2 -15309.656} C_VEL
LIN {X 0,Y 321.522,Z 867.857,A -85,B 0,C 180,E1 -15311.665,E2 -15311.665} C_VEL
LIN {X 0,Y 322.252,Z 857.934,A -85,B 0,C 180,E1 -15313.559,E2 -15313.559} C_VEL
LIN {X 0,Y 323.194,Z 846.771,A -85,B 0,C 180,E1 -15315.288,E2 -15315.288} C_VEL
LIN {X 0,Y 324.062,Z 834.941,A -85,B 0,C 180,E1 -15316.766,E2 -15316.766} C_VEL
LIN {X 0,Y 324.244,Z 831.389,A -85,B 0,C 180,E1 -15317.148,E2 -15317.148} C_VEL
LIN {X 0,Y 321.114,Z 818.696,A -85,B 0,C 180,E1 -15318.482,E2 -15318.482} C_VEL
LIN {X 0,Y 319.581,Z 812.675,A -85,B 0,C 180,E1 -15319.036,E2 -15319.036} C_VEL
LIN {X 0,Y 319.584,Z 812.67,A -85,B 0,C 180,E1 -15322.534,E2 -15322.534} C_VEL
LIN {X 0,Y 319.555,Z 812.672,A -85,B 0,C 180,E1 -15326.095,E2 -15326.095} C_VEL
LIN {X 0,Y 319.531,Z 812.676,A -85,B 0,C 180,E1 -15328.94,E2 -15328.94} C_VEL
LIN {X 0,Y 319.531,Z 812.674,A -85,B 0,C 180,E1 -15331.862,E2 -15331.862} C_VEL
LIN {X 0,Y 319.585,Z 812.674,A -85,B 0,C 180,E1 -15335.542,E2 -15335.542} C_VEL
LIN {X 0,Y 319.535,Z 812.68,A -85,B 0,C 180,E1 -15339.661,E2 -15339.661} C_VEL
LIN {X 0,Y 319.527,Z 812.679,A -85,B 0,C 180,E1 -15343.459,E2 -15343.459} C_VEL
LIN {X 0,Y 319.559,Z 812.676,A -85,B 0,C 180,E1 -15347.015,E2 -15347.015} C_VEL
LIN {X 0,Y 319.552,Z 812.679,A -85,B 0,C 180,E1 -15350.369,E2 -15350.369} C_VEL
LIN {X 0,Y 319.586,Z 812.677,A -85,B 0,C 180,E1 -15354.456,E2 -15354.456} C_VEL
LIN {X 0,Y 319.537,Z 812.678,A -85,B 0,C 180,E1 -15358.137,E2 -15358.137} C_VEL
LIN {X 0,Y 319.617,Z 812.664,A -85,B 0,C 180,E1 -15361.589,E2 -15361.589} C_VEL
LIN {X 0,Y 319.611,Z 812.661,A -85,B 0,C 180,E1 -15365.302,E2 -15365.302} C_VEL
LIN {X 0,Y 319.635,Z 812.67,A -85,B 0,C 180,E1 -15368.011,E2 -15368.011} C_VEL
LIN {X 0,Y 324.574,Z 826.608,A -85,B 0,C 180,E1 -15369.472,E2 -15369.472} C_VEL
LIN {X 0,Y 327.63,Z 836.654,A -85,B 0,C 180,E1 -15370.708,E2 -15370.708} C_VEL
LIN {X 0,Y 328.145,Z 839.673,A -85,B 0,C 180,E1 -15371.098,E2 -15371.098} C_VEL
LIN {X 0,Y 327.006,Z 849.696,A -85,B 0,C 180,E1 -15372.326,E2 -15372.326} C_VEL
LIN {X 0,Y 325.913,Z 858.879,A -85,B 0,C 180,E1 -15373.718,E2 -15373.718} C_VEL
LIN {X 0,Y 324.784,Z 867.24,A -85,B 0,C 180,E1 -15375.268,E2 -15375.268} C_VEL
LIN {X 0,Y 323.496,Z 875.358,A -85,B 0,C 180,E1 -15377.131,E2 -15377.131} C_VEL
LIN {X 0,Y 322.701,Z 880.886,A -85,B 0,C 180,E1 -15378.694,E2 -15378.694} C_VEL
LIN {X 0,Y 321.902,Z 886.265,A -85,B 0,C 180,E1 -15380.574,E2 -15380.574} C_VEL
LIN {X 0,Y 320.937,Z 890.529,A -85,B 0,C 180,E1 -15382.448,E2 -15382.448} C_VEL
LIN {X 0,Y 320.589,Z 892.755,A -85,B 0,C 180,E1 -15383.705,E2 -15383.705} C_VEL
LIN {X 0,Y 320.277,Z 894.571,A -85,B 0,C 180,E1 -15384.962,E2 -15384.962} C_VEL
LIN {X 0,Y 320.269,Z 895.906,A -85,B 0,C 180,E1 -15386.223,E2 -15386.223} C_VEL
LIN {X 0,Y 319.951,Z 897.485,A -85,B 0,C 180,E1 -15388.739,E2 -15388.739} C_VEL
LIN {X 0,Y 319.902,Z 897.715,A -85,B 0,C 180,E1 -15389.998,E2 -15389.998} C_VEL
LIN {X 0,Y 320.092,Z 896.95,A -85,B 0,C 180,E1 -15392.515,E2 -15392.515} C_VEL
LIN {X 0,Y 320.232,Z 896.01,A -85,B 0,C 180,E1 -15393.773,E2 -15393.773} C_VEL
LIN {X 0,Y 320.264,Z 894.716,A -85,B 0,C 180,E1 -15395.033,E2 -15395.033} C_VEL
LIN {X 0,Y 320.755,Z 891.91,A -85,B 0,C 180,E1 -15396.919,E2 -15396.919} C_VEL
LIN {X 0,Y 321.635,Z 888.069,A -85,B 0,C 180,E1 -15398.796,E2 -15398.796} C_VEL
LIN {X 0,Y 322.451,Z 883.158,A -85,B 0,C 180,E1 -15400.674,E2 -15400.674} C_VEL
LIN {X 0,Y 323.241,Z 876.991,A -85,B 0,C 180,E1 -15402.555,E2 -15402.555} C_VEL
LIN {X 0,Y 324.487,Z 869.215,A -85,B 0,C 180,E1 -15404.42,E2 -15404.42} C_VEL
LIN {X 0,Y 325.605,Z 861.285,A -85,B 0,C 180,E1 -15405.971,E2 -15405.971} C_VEL
LIN {X 0,Y 326.838,Z 851.591,A -85,B 0,C 180,E1 -15407.518,E2 -15407.518} C_VEL
LIN {X 0,Y 327.921,Z 842.032,A -85,B 0,C 180,E1 -15408.75,E2 -15408.75} C_VEL
LIN {X 0,Y 328.22,Z 838.897,A -85,B 0,C 180,E1 -15409.098,E2 -15409.098} C_VEL
LIN {X 0,Y 325.084,Z 827.974,A -85,B 0,C 180,E1 -15410.48,E2 -15410.48} C_VEL
LIN {X 0,Y 321.123,Z 817.037,A -85,B 0,C 180,E1 -15411.671,E2 -15411.671} C_VEL
LIN {X 0,Y 319.621,Z 812.67,A -85,B 0,C 180,E1 -15412.097,E2 -15412.097} C_VEL
LIN {X 0,Y 319.63,Z 812.672,A -85,B 0,C 180,E1 -15416.085,E2 -15416.085} C_VEL
LIN {X 0,Y 319.584,Z 812.676,A -85,B 0,C 180,E1 -15418.931,E2 -15418.931} C_VEL
LIN {X 0,Y 319.527,Z 812.686,A -85,B 0,C 180,E1 -15421.859,E2 -15421.859} C_VEL
LIN {X 0,Y 319.573,Z 812.678,A -85,B 0,C 180,E1 -15425.541,E2 -15425.541} C_VEL
LIN {X 0,Y 319.592,Z 812.677,A -85,B 0,C 180,E1 -15428.002,E2 -15428.002} C_VEL
LIN {X 0,Y 319.593,Z 812.674,A -85,B 0,C 180,E1 -15431.61,E2 -15431.61} C_VEL
LIN {X 0,Y 319.636,Z 812.668,A -85,B 0,C 180,E1 -15435.283,E2 -15435.283} C_VEL
LIN {X 0,Y 319.573,Z 812.679,A -85,B 0,C 180,E1 -15438.718,E2 -15438.718} C_VEL
LIN {X 0,Y 319.589,Z 812.672,A -85,B 0,C 180,E1 -15442.337,E2 -15442.337} C_VEL
LIN {X 0,Y 319.548,Z 812.673,A -85,B 0,C 180,E1 -15445.122,E2 -15445.122} C_VEL
LIN {X 0,Y 319.557,Z 812.675,A -85,B 0,C 180,E1 -15449.056,E2 -15449.056} C_VEL
LIN {X 0,Y 319.595,Z 812.675,A -85,B 0,C 180,E1 -15452.497,E2 -15452.497} C_VEL
LIN {X 0,Y 319.592,Z 812.669,A -85,B 0,C 180,E1 -15453.478,E2 -15453.478} C_VEL
LIN {X 0,Y 318.965,Z 812.749,A -85,B 0,C 180,E1 -15454.53,E2 -15454.53} C_VEL
LIN {X 0,Y 316.123,Z 813.107,A -85,B 0,C 180,E1 -15456.242,E2 -15456.242} C_VEL
LIN {X 0,Y 313.684,Z 813.412,A -85,B 0,C 180,E1 -15457.63,E2 -15457.63} C_VEL
LIN {X 0,Y 312.626,Z 813.54,A -85,B 0,C 180,E1 -15458.705,E2 -15458.705} C_VEL
LIN {X 0,Y 312.535,Z 813.549,A -85,B 0,C 180,E1 -15459.069,E2 -15459.069} C_VEL
LIN {X 0,Y 312.623,Z 813.542,A -85,B 0,C 180,E1 -15461.655,E2 -15461.655} C_VEL
LIN {X 0,Y 312.678,Z 813.533,A -85,B 0,C 180,E1 -15465.685,E2 -15465.685} C_VEL
LIN {X 0,Y 312.687,Z 813.531,A -85,B 0,C 180,E1 -15469.641,E2 -15469.641} C_VEL
LIN {X 0,Y 312.849,Z 813.513,A -85,B 0,C 180,E1 -15472.254,E2 -15472.254} C_VEL
LIN {X 0,Y 312.699,Z 813.537,A -85,B 0,C 180,E1 -15474.842,E2 -15474.842} C_VEL
LIN {X 0,Y 312.976,Z 813.5,A -85,B 0,C 180,E1 -15478.713,E2 -15478.713} C_VEL
LIN {X 0,Y 312.973,Z 813.503,A -85,B 0,C 180,E1 -15481.287,E2 -15481.287} C_VEL
LIN {X 0,Y 312.692,Z 813.537,A -85,B 0,C 180,E1 -15485.158,E2 -15485.158} C_VEL
LIN {X 0,Y 312.845,Z 813.519,A -85,B 0,C 180,E1 -15487.746,E2 -15487.746} C_VEL
LIN {X 0,Y 312.655,Z 813.535,A -85,B 0,C 180,E1 -15491.672,E2 -15491.672} C_VEL
LIN {X 0,Y 312.684,Z 813.535,A -85,B 0,C 180,E1 -15494.888,E2 -15494.888} C_VEL
LIN {X 0,Y 312.593,Z 813.548,A -85,B 0,C 180,E1 -15499.226,E2 -15499.226} C_VEL
LIN {X 0,Y 312.506,Z 813.558,A -85,B 0,C 180,E1 -15502.78,E2 -15502.78} C_VEL
LIN {X 0,Y 312.514,Z 813.558,A -85,B 0,C 180,E1 -15505.909,E2 -15505.909} C_VEL
LIN {X 0,Y 312.481,Z 813.562,A -85,B 0,C 180,E1 -15509.657,E2 -15509.657} C_VEL
LIN {X 0,Y 312.506,Z 813.558,A -85,B 0,C 180,E1 -15513.69,E2 -15513.69} C_VEL
LIN {X 0,Y 312.496,Z 813.56,A -85,B 0,C 180,E1 -15517.389,E2 -15517.389} C_VEL
LIN {X 0,Y 312.49,Z 813.64,A -85,B 0,C 180,E1 -15520.186,E2 -15520.186} C_VEL
LIN {X 0,Y 314.095,Z 821.174,A -85,B 0,C 180,E1 -15523.919,E2 -15523.919} C_VEL
LIN {X 0,Y 315.557,Z 828.496,A -85,B 0,C 180,E1 -15527.305,E2 -15527.305} C_VEL
LIN {X 0,Y 317.068,Z 836.765,A -85,B 0,C 180,E1 -15530.877,E2 -15530.877} C_VEL
LIN {X 0,Y 317.281,Z 840.49,A -85,B 0,C 180,E1 -15532.391,E2 -15532.391} C_VEL
LIN {X 0,Y 315.523,Z 852.435,A -85,B 0,C 180,E1 -15536.93,E2 -15536.93} C_VEL
LIN {X 0,Y 314.057,Z 864.207,A -85,B 0,C 180,E1 -15541.338,E2 -15541.338} C_VEL
LIN {X 0,Y 312.924,Z 875.216,A -85,B 0,C 180,E1 -15545.453,E2 -15545.453} C_VEL
LIN {X 0,Y 312.676,Z 878.094,A -85,B 0,C 180,E1 -15546.545,E2 -15546.545} C_VEL
LIN {X 0,Y 314.92,Z 893.319,A -85,B 0,C 180,E1 -15547.311,E2 -15547.311} C_VEL
LIN {X 0,Y 316.147,Z 906.678,A -85,B 0,C 180,E1 -15548.214,E2 -15548.214} C_VEL
LIN {X 0,Y 316.598,Z 918.269,A -85,B 0,C 180,E1 -15549.199,E2 -15549.199} C_VEL
LIN {X 0,Y 316.487,Z 931.049,A -85,B 0,C 180,E1 -15550.546,E2 -15550.546} C_VEL
LIN {X 0,Y 316.366,Z 938.796,A -85,B 0,C 180,E1 -15551.548,E2 -15551.548} C_VEL
LIN {X 0,Y 314.846,Z 949.429,A -85,B 0,C 180,E1 -15553.134,E2 -15553.134} C_VEL
LIN {X 0,Y 313.414,Z 958.342,A -85,B 0,C 180,E1 -15554.79,E2 -15554.79} C_VEL
LIN {X 0,Y 312.92,Z 963.935,A -85,B 0,C 180,E1 -15556.031,E2 -15556.031} C_VEL
LIN {X 0,Y 312.14,Z 971.343,A -85,B 0,C 180,E1 -15557.982,E2 -15557.982} C_VEL
LIN {X 0,Y 311.656,Z 978.14,A -85,B 0,C 180,E1 -15560.265,E2 -15560.265} C_VEL
LIN {X 0,Y 311.547,Z 982.677,A -85,B 0,C 180,E1 -15562.224,E2 -15562.224} C_VEL
LIN {X 0,Y 311.618,Z 985.102,A -85,B 0,C 180,E1 -15563.528,E2 -15563.528} C_VEL
LIN {X 0,Y 311.768,Z 987.079,A -85,B 0,C 180,E1 -15564.829,E2 -15564.829} C_VEL
LIN {X 0,Y 311.92,Z 988.569,A -85,B 0,C 180,E1 -15566.127,E2 -15566.127} C_VEL
LIN {X 0,Y 311.974,Z 989.622,A -85,B 0,C 180,E1 -15567.42,E2 -15567.42} C_VEL
LIN {X 0,Y 312.072,Z 990.273,A -85,B 0,C 180,E1 -15568.712,E2 -15568.712} C_VEL
LIN {X 0,Y 312.16,Z 990.509,A -85,B 0,C 180,E1 -15570.002,E2 -15570.002} C_VEL
LIN {X 0,Y 312.073,Z 990.266,A -85,B 0,C 180,E1 -15571.293,E2 -15571.293} C_VEL
LIN {X 0,Y 311.975,Z 989.609,A -85,B 0,C 180,E1 -15572.585,E2 -15572.585} C_VEL
LIN {X 0,Y 311.921,Z 988.55,A -85,B 0,C 180,E1 -15573.878,E2 -15573.878} C_VEL
LIN {X 0,Y 311.77,Z 987.054,A -85,B 0,C 180,E1 -15575.176,E2 -15575.176} C_VEL
LIN {X 0,Y 311.628,Z 983.978,A -85,B 0,C 180,E1 -15577.108,E2 -15577.108} C_VEL
LIN {X 0,Y 311.583,Z 979.76,A -85,B 0,C 180,E1 -15579.087,E2 -15579.087} C_VEL
LIN {X 0,Y 311.914,Z 973.385,A -85,B 0,C 180,E1 -15581.373,E2 -15581.373} C_VEL
LIN {X 0,Y 312.935,Z 964.135,A -85,B 0,C 180,E1 -15583.973,E2 -15583.973} C_VEL
LIN {X 0,Y 314.033,Z 956.697,A -85,B 0,C 180,E1 -15585.776,E2 -15585.776} C_VEL
LIN {X 0,Y 315.796,Z 946.55,A -85,B 0,C 180,E1 -15587.821,E2 -15587.821} C_VEL
LIN {X 0,Y 317.204,Z 938.942,A -85,B 0,C 180,E1 -15589.077,E2 -15589.077} C_VEL
LIN {X 0,Y 317.736,Z 930.515,A -85,B 0,C 180,E1 -15590.39,E2 -15590.39} C_VEL
LIN {X 0,Y 318.661,Z 919.242,A -85,B 0,C 180,E1 -15591.887,E2 -15591.887} C_VEL
LIN {X 0,Y 319.257,Z 909.697,A -85,B 0,C 180,E1 -15593.002,E2 -15593.002} C_VEL
LIN {X 0,Y 318.802,Z 898.727,A -85,B 0,C 180,E1 -15594.245,E2 -15594.245} C_VEL
LIN {X 0,Y 317.459,Z 886.653,A -85,B 0,C 180,E1 -15595.565,E2 -15595.565} C_VEL
LIN {X 0,Y 315.641,Z 876.27,A -85,B 0,C 180,E1 -15596.708,E2 -15596.708} C_VEL
LIN {X 0,Y 314.766,Z 871.91,A -85,B 0,C 180,E1 -15597.173,E2 -15597.173} C_VEL
LIN {X 0,Y 313.839,Z 867.296,A -85,B 0,C 180,E1 -15597.682,E2 -15597.682} C_VEL
LIN {X 0,Y 313.834,Z 866.543,A -85,B 0,C 180,E1 -15597.775,E2 -15597.775} C_VEL
LIN {X 0,Y 315.237,Z 854.304,A -85,B 0,C 180,E1 -15602.35,E2 -15602.35} C_VEL
LIN {X 0,Y 316.604,Z 844.54,A -85,B 0,C 180,E1 -15606.035,E2 -15606.035} C_VEL
LIN {X 0,Y 317.28,Z 840.403,A -85,B 0,C 180,E1 -15607.616,E2 -15607.616} C_VEL
LIN {X 0,Y 317.058,Z 836.704,A -85,B 0,C 180,E1 -15609.12,E2 -15609.12} C_VEL
LIN {X 0,Y 315.518,Z 828.461,A -85,B 0,C 180,E1 -15612.688,E2 -15612.688} C_VEL
LIN {X 0,Y 314.039,Z 821.055,A -85,B 0,C 180,E1 -15616.071,E2 -15616.071} C_VEL
LIN {X 0,Y 312.491,Z 813.56,A -85,B 0,C 180,E1 -15619.88,E2 -15619.88} C_VEL
LIN {X 0,Y 312.538,Z 813.553,A -85,B 0,C 180,E1 -15624.052,E2 -15624.052} C_VEL
LIN {X 0,Y 312.507,Z 813.556,A -85,B 0,C 180,E1 -15627.334,E2 -15627.334} C_VEL
LIN {X 0,Y 312.518,Z 813.555,A -85,B 0,C 180,E1 -15631.493,E2 -15631.493} C_VEL
LIN {X 0,Y 313.172,Z 815.807,A -85,B 0,C 180,E1 -15631.883,E2 -15631.883} C_VEL
LIN {X 0,Y 318.151,Z 823.362,A -85,B 0,C 180,E1 -15633.781,E2 -15633.781} C_VEL
LIN {X 0,Y 322.693,Z 832.709,A -85,B 0,C 180,E1 -15635.774,E2 -15635.774} C_VEL
LIN {X 0,Y 325.698,Z 840.622,A -85,B 0,C 180,E1 -15637.358,E2 -15637.358} C_VEL
LIN {X 0,Y 327.476,Z 847.048,A -85,B 0,C 180,E1 -15638.602,E2 -15638.602} C_VEL
LIN {X 0,Y 327.749,Z 848.704,A -85,B 0,C 180,E1 -15638.914,E2 -15638.914} C_VEL
LIN {X 0,Y 326.161,Z 857.321,A -85,B 0,C 180,E1 -15640.161,E2 -15640.161} C_VEL
LIN {X 0,Y 324.62,Z 864.497,A -85,B 0,C 180,E1 -15641.377,E2 -15641.377} C_VEL
LIN {X 0,Y 322.876,Z 872.185,A -85,B 0,C 180,E1 -15642.911,E2 -15642.911} C_VEL
LIN {X 0,Y 320.624,Z 880.921,A -85,B 0,C 180,E1 -15645.122,E2 -15645.122} C_VEL
LIN {X 0,Y 318.703,Z 887.342,A -85,B 0,C 180,E1 -15647.26,E2 -15647.26} C_VEL
LIN {X 0,Y 317.245,Z 891.813,A -85,B 0,C 180,E1 -15649.146,E2 -15649.146} C_VEL
LIN {X 0,Y 315.992,Z 895.055,A -85,B 0,C 180,E1 -15651.043,E2 -15651.043} C_VEL
LIN {X 0,Y 315.202,Z 896.813,A -85,B 0,C 180,E1 -15652.312,E2 -15652.312} C_VEL
LIN {X 0,Y 314.262,Z 898.718,A -85,B 0,C 180,E1 -15654.868,E2 -15654.868} C_VEL
LIN {X 0,Y 313.882,Z 899.199,A -85,B 0,C 180,E1 -15656.148,E2 -15656.148} C_VEL
LIN {X 0,Y 313.22,Z 898.762,A -85,B 0,C 180,E1 -15658.714,E2 -15658.714} C_VEL
LIN {X 0,Y 312.876,Z 897.971,A -85,B 0,C 180,E1 -15660,E2 -15660} C_VEL
LIN {X 0,Y 312.731,Z 894.966,A -85,B 0,C 180,E1 -15662.576,E2 -15662.576} C_VEL
LIN {X 0,Y 312.593,Z 892.958,A -85,B 0,C 180,E1 -15663.868,E2 -15663.868} C_VEL
LIN {X 0,Y 313.004,Z 888.909,A -85,B 0,C 180,E1 -15665.799,E2 -15665.799} C_VEL
LIN {X 0,Y 313.435,Z 882.698,A -85,B 0,C 180,E1 -15668.056,E2 -15668.056} C_VEL
LIN {X 0,Y 313.785,Z 876.918,A -85,B 0,C 180,E1 -15669.764,E2 -15669.764} C_VEL
LIN {X 0,Y 314.421,Z 869.426,A -85,B 0,C 180,E1 -15671.605,E2 -15671.605} C_VEL
LIN {X 0,Y 315.059,Z 861.34,A -85,B 0,C 180,E1 -15673.217,E2 -15673.217} C_VEL
LIN {X 0,Y 315.619,Z 853.834,A -85,B 0,C 180,E1 -15674.508,E2 -15674.508} C_VEL
LIN {X 0,Y 316.336,Z 845.057,A -85,B 0,C 180,E1 -15675.793,E2 -15675.793} C_VEL
LIN {X 0,Y 317.076,Z 835.865,A -85,B 0,C 180,E1 -15676.949,E2 -15676.949} C_VEL
LIN {X 0,Y 317.22,Z 832.254,A -85,B 0,C 180,E1 -15677.346,E2 -15677.346} C_VEL
LIN {X 0,Y 314.034,Z 819.561,A -85,B 0,C 180,E1 -15678.707,E2 -15678.707} C_VEL
LIN {X 0,Y 312.531,Z 813.555,A -85,B 0,C 180,E1 -15679.283,E2 -15679.283} C_VEL
LIN {X 0,Y 312.516,Z 813.55,A -85,B 0,C 180,E1 -15682.772,E2 -15682.772} C_VEL
LIN {X 0,Y 312.488,Z 813.549,A -85,B 0,C 180,E1 -15686.732,E2 -15686.732} C_VEL
LIN {X 0,Y 312.476,Z 813.559,A -85,B 0,C 180,E1 -15689.657,E2 -15689.657} C_VEL
LIN {X 0,Y 312.527,Z 813.546,A -85,B 0,C 180,E1 -15693.688,E2 -15693.688} C_VEL
LIN {X 0,Y 312.516,Z 813.549,A -85,B 0,C 180,E1 -15697.387,E2 -15697.387} C_VEL
LIN {X 0,Y 312.448,Z 813.561,A -85,B 0,C 180,E1 -15700.716,E2 -15700.716} C_VEL
LIN {X 0,Y 312.458,Z 813.565,A -85,B 0,C 180,E1 -15704.209,E2 -15704.209} C_VEL
LIN {X 0,Y 312.462,Z 813.564,A -85,B 0,C 180,E1 -15707.923,E2 -15707.923} C_VEL
LIN {X 0,Y 312.484,Z 813.563,A -85,B 0,C 180,E1 -15711.923,E2 -15711.923} C_VEL
LIN {X 0,Y 312.538,Z 813.555,A -85,B 0,C 180,E1 -15714.219,E2 -15714.219} C_VEL
LIN {X 0,Y 312.51,Z 813.554,A -85,B 0,C 180,E1 -15717.332,E2 -15717.332} C_VEL
LIN {X 0,Y 312.551,Z 813.544,A -85,B 0,C 180,E1 -15721.277,E2 -15721.277} C_VEL
LIN {X 0,Y 312.592,Z 813.538,A -85,B 0,C 180,E1 -15724.709,E2 -15724.709} C_VEL
LIN {X 0,Y 312.603,Z 813.712,A -85,B 0,C 180,E1 -15727.506,E2 -15727.506} C_VEL
LIN {X 0,Y 316.801,Z 825.159,A -85,B 0,C 180,E1 -15728.709,E2 -15728.709} C_VEL
LIN {X 0,Y 320.207,Z 835.775,A -85,B 0,C 180,E1 -15730.02,E2 -15730.02} C_VEL
LIN {X 0,Y 321.483,Z 840.713,A -85,B 0,C 180,E1 -15730.691,E2 -15730.691} C_VEL
LIN {X 0,Y 320.192,Z 851.875,A -85,B 0,C 180,E1 -15732.102,E2 -15732.102} C_VEL
LIN {X 0,Y 318.943,Z 861.696,A -85,B 0,C 180,E1 -15733.681,E2 -15733.681} C_VEL
LIN {X 0,Y 317.742,Z 869.732,A -85,B 0,C 180,E1 -15735.262,E2 -15735.262} C_VEL
LIN {X 0,Y 316.42,Z 877.597,A -85,B 0,C 180,E1 -15737.165,E2 -15737.165} C_VEL
LIN {X 0,Y 315.56,Z 883.866,A -85,B 0,C 180,E1 -15739.085,E2 -15739.085} C_VEL
LIN {X 0,Y 314.675,Z 888.859,A -85,B 0,C 180,E1 -15741.003,E2 -15741.003} C_VEL
LIN {X 0,Y 313.795,Z 892.752,A -85,B 0,C 180,E1 -15742.922,E2 -15742.922} C_VEL
LIN {X 0,Y 313.28,Z 895.604,A -85,B 0,C 180,E1 -15744.849,E2 -15744.849} C_VEL
LIN {X 0,Y 313.266,Z 896.937,A -85,B 0,C 180,E1 -15746.139,E2 -15746.139} C_VEL
LIN {X 0,Y 312.929,Z 898.516,A -85,B 0,C 180,E1 -15748.711,E2 -15748.711} C_VEL
LIN {X 0,Y 312.878,Z 898.746,A -85,B 0,C 180,E1 -15749.998,E2 -15749.998} C_VEL
LIN {X 0,Y 313.078,Z 897.98,A -85,B 0,C 180,E1 -15752.571,E2 -15752.571} C_VEL
LIN {X 0,Y 313.234,Z 897.04,A -85,B 0,C 180,E1 -15753.857,E2 -15753.857} C_VEL
LIN {X 0,Y 313.267,Z 895.746,A -85,B 0,C 180,E1 -15755.146,E2 -15755.146} C_VEL
LIN {X 0,Y 313.782,Z 892.94,A -85,B 0,C 180,E1 -15757.074,E2 -15757.074} C_VEL
LIN {X 0,Y 314.696,Z 889.098,A -85,B 0,C 180,E1 -15758.991,E2 -15758.991} C_VEL
LIN {X 0,Y 315.552,Z 884.187,A -85,B 0,C 180,E1 -15760.91,E2 -15760.91} C_VEL
LIN {X 0,Y 316.388,Z 878.021,A -85,B 0,C 180,E1 -15762.832,E2 -15762.832} C_VEL
LIN {X 0,Y 317.689,Z 870.243,A -85,B 0,C 180,E1 -15764.736,E2 -15764.736} C_VEL
LIN {X 0,Y 318.857,Z 862.313,A -85,B 0,C 180,E1 -15766.319,E2 -15766.319} C_VEL
LIN {X 0,Y 320.147,Z 852.619,A -85,B 0,C 180,E1 -15767.896,E2 -15767.896} C_VEL
LIN {X 0,Y 321.283,Z 843.057,A -85,B 0,C 180,E1 -15769.152,E2 -15769.152} C_VEL
LIN {X 0,Y 321.428,Z 840.25,A -85,B 0,C 180,E1 -15769.481,E2 -15769.481} C_VEL
LIN {X 0,Y 318.613,Z 830.42,A -85,B 0,C 180,E1 -15770.774,E2 -15770.774} C_VEL
LIN {X 0,Y 314.802,Z 819.646,A -85,B 0,C 180,E1 -15772.014,E2 -15772.014} C_VEL
LIN {X 0,Y 312.563,Z 813.548,A -85,B 0,C 180,E1 -15772.645,E2 -15772.645} C_VEL
LIN {X 0,Y 312.599,Z 813.548,A -85,B 0,C 180,E1 -15775.933,E2 -15775.933} C_VEL
LIN {X 0,Y 312.54,Z 813.555,A -85,B 0,C 180,E1 -15779.647,E2 -15779.647} C_VEL
LIN {X 0,Y 312.513,Z 813.558,A -85,B 0,C 180,E1 -15783.686,E2 -15783.686} C_VEL
LIN {X 0,Y 312.545,Z 813.553,A -85,B 0,C 180,E1 -15787.379,E2 -15787.379} C_VEL
LIN {X 0,Y 312.527,Z 813.555,A -85,B 0,C 180,E1 -15790.7,E2 -15790.7} C_VEL
LIN {X 0,Y 312.585,Z 813.55,A -85,B 0,C 180,E1 -15794.182,E2 -15794.182} C_VEL
LIN {X 0,Y 312.546,Z 813.547,A -85,B 0,C 180,E1 -15797.902,E2 -15797.902} C_VEL
LIN {X 0,Y 312.549,Z 813.546,A -85,B 0,C 180,E1 -15801.902,E2 -15801.902} C_VEL
LIN {X 0,Y 312.494,Z 813.551,A -85,B 0,C 180,E1 -15805.788,E2 -15805.788} C_VEL
LIN {X 0,Y 312.51,Z 813.554,A -85,B 0,C 180,E1 -15808.852,E2 -15808.852} C_VEL
LIN {X 0,Y 312.561,Z 813.548,A -85,B 0,C 180,E1 -15811.823,E2 -15811.823} C_VEL
LIN {X 0,Y 312.571,Z 813.545,A -85,B 0,C 180,E1 -15814.709,E2 -15814.709} C_VEL
LIN {X 0,Y 312.572,Z 813.547,A -85,B 0,C 180,E1 -15817.528,E2 -15817.528} C_VEL
LIN {X 0,Y 312.535,Z 813.549,A -85,B 0,C 180,E1 -15819.069,E2 -15819.069} C_VEL
LIN {X 0,Y 311.854,Z 813.634,A -85,B 0,C 180,E1 -15820.145,E2 -15820.145} C_VEL
LIN {X 0,Y 309.007,Z 813.991,A -85,B 0,C 180,E1 -15821.898,E2 -15821.898} C_VEL
LIN {X 0,Y 306.635,Z 814.284,A -85,B 0,C 180,E1 -15823.319,E2 -15823.319} C_VEL
LIN {X 0,Y 305.663,Z 814.401,A -85,B 0,C 180,E1 -15824.42,E2 -15824.42} C_VEL
LIN {X 0,Y 305.608,Z 814.407,A -85,B 0,C 180,E1 -15824.792,E2 -15824.792} C_VEL
LIN {X 0,Y 305.591,Z 814.419,A -85,B 0,C 180,E1 -15828.054,E2 -15828.054} C_VEL
LIN {X 0,Y 305.792,Z 814.393,A -85,B 0,C 180,E1 -15832.074,E2 -15832.074} C_VEL
LIN {X 0,Y 305.67,Z 814.412,A -85,B 0,C 180,E1 -15834.723,E2 -15834.723} C_VEL
LIN {X 0,Y 305.942,Z 814.376,A -85,B 0,C 180,E1 -15838.684,E2 -15838.684} C_VEL
LIN {X 0,Y 305.94,Z 814.38,A -85,B 0,C 180,E1 -15841.316,E2 -15841.316} C_VEL
LIN {X 0,Y 305.662,Z 814.413,A -85,B 0,C 180,E1 -15845.277,E2 -15845.277} C_VEL
LIN {X 0,Y 305.788,Z 814.396,A -85,B 0,C 180,E1 -15847.926,E2 -15847.926} C_VEL
LIN {X 0,Y 305.589,Z 814.413,A -85,B 0,C 180,E1 -15851.946,E2 -15851.946} C_VEL
LIN {X 0,Y 305.622,Z 814.415,A -85,B 0,C 180,E1 -15855.036,E2 -15855.036} C_VEL
LIN {X 0,Y 305.564,Z 814.423,A -85,B 0,C 180,E1 -15858.784,E2 -15858.784} C_VEL
LIN {X 0,Y 305.471,Z 814.434,A -85,B 0,C 180,E1 -15863.041,E2 -15863.041} C_VEL
LIN {X 0,Y 305.454,Z 814.437,A -85,B 0,C 180,E1 -15866.198,E2 -15866.198} C_VEL
LIN {X 0,Y 305.434,Z 814.439,A -85,B 0,C 180,E1 -15869.035,E2 -15869.035} C_VEL
LIN {X 0,Y 305.422,Z 814.441,A -85,B 0,C 180,E1 -15871.955,E2 -15871.955} C_VEL
LIN {X 0,Y 305.447,Z 814.436,A -85,B 0,C 180,E1 -15875.115,E2 -15875.115} C_VEL
LIN {X 0,Y 305.429,Z 814.442,A -85,B 0,C 180,E1 -15879.256,E2 -15879.256} C_VEL
LIN {X 0,Y 305.453,Z 814.657,A -85,B 0,C 180,E1 -15879.679,E2 -15879.679} C_VEL
LIN {X 0,Y 307.018,Z 821.868,A -85,B 0,C 180,E1 -15883.372,E2 -15883.372} C_VEL
LIN {X 0,Y 308.485,Z 829.275,A -85,B 0,C 180,E1 -15886.889,E2 -15886.889} C_VEL
LIN {X 0,Y 309.653,Z 835.521,A -85,B 0,C 180,E1 -15889.694,E2 -15889.694} C_VEL
LIN {X 0,Y 310.329,Z 840.671,A -85,B 0,C 180,E1 -15891.897,E2 -15891.897} C_VEL
LIN {X 0,Y 309.054,Z 849.468,A -85,B 0,C 180,E1 -15895.357,E2 -15895.357} C_VEL
LIN {X 0,Y 307.456,Z 861.004,A -85,B 0,C 180,E1 -15899.812,E2 -15899.812} C_VEL
LIN {X 0,Y 306.181,Z 872.282,A -85,B 0,C 180,E1 -15904.146,E2 -15904.146} C_VEL
LIN {X 0,Y 305.707,Z 877.155,A -85,B 0,C 180,E1 -15906,E2 -15906} C_VEL
LIN {X 0,Y 307.912,Z 891.622,A -85,B 0,C 180,E1 -15906.736,E2 -15906.736} C_VEL
LIN {X 0,Y 309.115,Z 903.768,A -85,B 0,C 180,E1 -15907.556,E2 -15907.556} C_VEL
LIN {X 0,Y 309.679,Z 915.713,A -85,B 0,C 180,E1 -15908.57,E2 -15908.57} C_VEL
LIN {X 0,Y 309.669,Z 927.052,A -85,B 0,C 180,E1 -15909.754,E2 -15909.754} C_VEL
LIN {X 0,Y 309.422,Z 938.941,A -85,B 0,C 180,E1 -15911.29,E2 -15911.29} C_VEL
LIN {X 0,Y 307.968,Z 948.376,A -85,B 0,C 180,E1 -15912.745,E2 -15912.745} C_VEL
LIN {X 0,Y 306.66,Z 956.823,A -85,B 0,C 180,E1 -15914.339,E2 -15914.339} C_VEL
LIN {X 0,Y 305.775,Z 964.24,A -85,B 0,C 180,E1 -15916.037,E2 -15916.037} C_VEL
LIN {X 0,Y 305.009,Z 971.35,A -85,B 0,C 180,E1 -15918.034,E2 -15918.034} C_VEL
LIN {X 0,Y 304.619,Z 977.092,A -85,B 0,C 180,E1 -15920.038,E2 -15920.038} C_VEL
LIN {X 0,Y 304.5,Z 981.634,A -85,B 0,C 180,E1 -15922.042,E2 -15922.042} C_VEL
LIN {X 0,Y 304.558,Z 984.059,A -85,B 0,C 180,E1 -15923.377,E2 -15923.377} C_VEL
LIN {X 0,Y 304.7,Z 986.038,A -85,B 0,C 180,E1 -15924.709,E2 -15924.709} C_VEL
LIN {X 0,Y 304.876,Z 987.533,A -85,B 0,C 180,E1 -15926.037,E2 -15926.037} C_VEL
LIN {X 0,Y 304.933,Z 988.587,A -85,B 0,C 180,E1 -15927.36,E2 -15927.36} C_VEL
LIN {X 0,Y 305.037,Z 989.24,A -85,B 0,C 180,E1 -15928.682,E2 -15928.682} C_VEL
LIN {X 0,Y 305.134,Z 989.477,A -85,B 0,C 180,E1 -15930.002,E2 -15930.002} C_VEL
LIN {X 0,Y 305.038,Z 989.232,A -85,B 0,C 180,E1 -15931.323,E2 -15931.323} C_VEL
LIN {X 0,Y 304.934,Z 988.574,A -85,B 0,C 180,E1 -15932.644,E2 -15932.644} C_VEL
LIN {X 0,Y 304.877,Z 987.513,A -85,B 0,C 180,E1 -15933.968,E2 -15933.968} C_VEL
LIN {X 0,Y 304.704,Z 986.011,A -85,B 0,C 180,E1 -15935.296,E2 -15935.296} C_VEL
LIN {X 0,Y 304.559,Z 983.18,A -85,B 0,C 180,E1 -15937.128,E2 -15937.128} C_VEL
LIN {X 0,Y 304.541,Z 978.712,A -85,B 0,C 180,E1 -15939.299,E2 -15939.299} C_VEL
LIN {X 0,Y 304.894,Z 972.35,A -85,B 0,C 180,E1 -15941.638,E2 -15941.638} C_VEL
LIN {X 0,Y 306.256,Z 962.506,A -85,B 0,C 180,E1 -15944.623,E2 -15944.623} C_VEL
LIN {X 0,Y 307.503,Z 954.727,A -85,B 0,C 180,E1 -15946.534,E2 -15946.534} C_VEL
LIN {X 0,Y 309.378,Z 944.917,A -85,B 0,C 180,E1 -15948.546,E2 -15948.546} C_VEL
LIN {X 0,Y 310.46,Z 939.365,A -85,B 0,C 180,E1 -15949.508,E2 -15949.508} C_VEL
LIN {X 0,Y 311.356,Z 929.009,A -85,B 0,C 180,E1 -15951.173,E2 -15951.173} C_VEL
LIN {X 0,Y 312.442,Z 917.54,A -85,B 0,C 180,E1 -15952.743,E2 -15952.743} C_VEL
LIN {X 0,Y 312.962,Z 908.636,A -85,B 0,C 180,E1 -15953.844,E2 -15953.844} C_VEL
LIN {X 0,Y 312.378,Z 895.297,A -85,B 0,C 180,E1 -15955.436,E2 -15955.436} C_VEL
LIN {X 0,Y 310.856,Z 883.07,A -85,B 0,C 180,E1 -15956.885,E2 -15956.885} C_VEL
LIN {X 0,Y 309.16,Z 873.647,A -85,B 0,C 180,E1 -15958.027,E2 -15958.027} C_VEL
LIN {X 0,Y 308.389,Z 869.537,A -85,B 0,C 180,E1 -15958.505,E2 -15958.505} C_VEL
LIN {X 0,Y 307.244,Z 864.718,A -85,B 0,C 180,E1 -15959.136,E2 -15959.136} C_VEL
LIN {X 0,Y 307.155,Z 863.291,A -85,B 0,C 180,E1 -15959.299,E2 -15959.299} C_VEL
LIN {X 0,Y 308.776,Z 851.332,A -85,B 0,C 180,E1 -15963.895,E2 -15963.895} C_VEL
LIN {X 0,Y 310.29,Z 841.583,A -85,B 0,C 180,E1 -15967.703,E2 -15967.703} C_VEL
LIN {X 0,Y 310,Z 837.522,A -85,B 0,C 180,E1 -15969.406,E2 -15969.406} C_VEL
LIN {X 0,Y 308.806,Z 830.967,A -85,B 0,C 180,E1 -15972.299,E2 -15972.299} C_VEL
LIN {X 0,Y 307.284,Z 823.332,A -85,B 0,C 180,E1 -15975.864,E2 -15975.864} C_VEL
LIN {X 0,Y 305.849,Z 816.528,A -85,B 0,C 180,E1 -15979.317,E2 -15979.317} C_VEL
LIN {X 0,Y 305.419,Z 814.442,A -85,B 0,C 180,E1 -15980.423,E2 -15980.423} C_VEL
LIN {X 0,Y 305.466,Z 814.432,A -85,B 0,C 180,E1 -15983.638,E2 -15983.638} C_VEL
LIN {X 0,Y 305.471,Z 814.436,A -85,B 0,C 180,E1 -15986.484,E2 -15986.484} C_VEL
LIN {X 0,Y 305.443,Z 814.532,A -85,B 0,C 180,E1 -15989.636,E2 -15989.636} C_VEL
LIN {X 0,Y 306.015,Z 816.52,A -85,B 0,C 180,E1 -15990.02,E2 -15990.02} C_VEL
LIN {X 0,Y 307.882,Z 818.978,A -85,B 0,C 180,E1 -15990.832,E2 -15990.832} C_VEL
LIN {X 0,Y 308.791,Z 820.024,A -85,B 0,C 180,E1 -15991.201,E2 -15991.201} C_VEL
LIN {X 0,Y 309.36,Z 821.42,A -85,B 0,C 180,E1 -15991.505,E2 -15991.505} C_VEL
LIN {X 0,Y 313.665,Z 828.413,A -85,B 0,C 180,E1 -15993.377,E2 -15993.377} C_VEL
LIN {X 0,Y 316.677,Z 834.886,A -85,B 0,C 180,E1 -15994.861,E2 -15994.861} C_VEL
LIN {X 0,Y 319.912,Z 843.343,A -85,B 0,C 180,E1 -15996.707,E2 -15996.707} C_VEL
LIN {X 0,Y 321.754,Z 850.552,A -85,B 0,C 180,E1 -15998.203,E2 -15998.203} C_VEL
LIN {X 0,Y 321.608,Z 852.953,A -85,B 0,C 180,E1 -15998.582,E2 -15998.582} C_VEL
LIN {X 0,Y 319.153,Z 864.146,A -85,B 0,C 180,E1 -16000.378,E2 -16000.378} C_VEL
LIN {X 0,Y 317.229,Z 872.02,A -85,B 0,C 180,E1 -16001.931,E2 -16001.931} C_VEL
LIN {X 0,Y 315.083,Z 879.542,A -85,B 0,C 180,E1 -16003.772,E2 -16003.772} C_VEL
LIN {X 0,Y 313.628,Z 884.538,A -85,B 0,C 180,E1 -16005.257,E2 -16005.257} C_VEL
LIN {X 0,Y 312.064,Z 889.348,A -85,B 0,C 180,E1 -16006.985,E2 -16006.985} C_VEL
LIN {X 0,Y 310.514,Z 893.669,A -85,B 0,C 180,E1 -16008.908,E2 -16008.908} C_VEL
LIN {X 0,Y 309.176,Z 896.725,A -85,B 0,C 180,E1 -16010.844,E2 -16010.844} C_VEL
LIN {X 0,Y 308.342,Z 898.345,A -85,B 0,C 180,E1 -16012.14,E2 -16012.14} C_VEL
LIN {X 0,Y 307.861,Z 899.442,A -85,B 0,C 180,E1 -16013.446,E2 -16013.446} C_VEL
LIN {X 0,Y 306.941,Z 900.469,A -85,B 0,C 180,E1 -16016.061,E2 -16016.061} C_VEL
LIN {X 0,Y 306.223,Z 899.886,A -85,B 0,C 180,E1 -16018.685,E2 -16018.685} C_VEL
LIN {X 0,Y 305.849,Z 898.974,A -85,B 0,C 180,E1 -16020,E2 -16020} C_VEL
LIN {X 0,Y 305.821,Z 897.576,A -85,B 0,C 180,E1 -16021.317,E2 -16021.317} C_VEL
LIN {X 0,Y 305.547,Z 893.683,A -85,B 0,C 180,E1 -16023.957,E2 -16023.957} C_VEL
LIN {X 0,Y 305.975,Z 889.473,A -85,B 0,C 180,E1 -16025.933,E2 -16025.933} C_VEL
LIN {X 0,Y 306.335,Z 884.136,A -85,B 0,C 180,E1 -16027.912,E2 -16027.912} C_VEL
LIN {X 0,Y 306.654,Z 879.204,A -85,B 0,C 180,E1 -16029.445,E2 -16029.445} C_VEL
LIN {X 0,Y 307.329,Z 870.947,A -85,B 0,C 180,E1 -16031.543,E2 -16031.543} C_VEL
LIN {X 0,Y 307.991,Z 862.953,A -85,B 0,C 180,E1 -16033.191,E2 -16033.191} C_VEL
LIN {X 0,Y 308.615,Z 854.517,A -85,B 0,C 180,E1 -16034.676,E2 -16034.676} C_VEL
LIN {X 0,Y 309.36,Z 845.676,A -85,B 0,C 180,E1 -16035.989,E2 -16035.989} C_VEL
LIN {X 0,Y 310.185,Z 835.045,A -85,B 0,C 180,E1 -16037.325,E2 -16037.325} C_VEL
LIN {X 0,Y 309.877,Z 831.706,A -85,B 0,C 180,E1 -16037.715,E2 -16037.715} C_VEL
LIN {X 0,Y 306.821,Z 819.786,A -85,B 0,C 180,E1 -16038.99,E2 -16038.99} C_VEL
LIN {X 0,Y 305.509,Z 814.427,A -85,B 0,C 180,E1 -16039.515,E2 -16039.515} C_VEL
LIN {X 0,Y 305.463,Z 814.429,A -85,B 0,C 180,E1 -16043.025,E2 -16043.025} C_VEL
LIN {X 0,Y 305.457,Z 814.427,A -85,B 0,C 180,E1 -16046.189,E2 -16046.189} C_VEL
LIN {X 0,Y 305.431,Z 814.432,A -85,B 0,C 180,E1 -16049.025,E2 -16049.025} C_VEL
LIN {X 0,Y 305.444,Z 814.428,A -85,B 0,C 180,E1 -16051.952,E2 -16051.952} C_VEL
LIN {X 0,Y 305.468,Z 814.43,A -85,B 0,C 180,E1 -16055.113,E2 -16055.113} C_VEL
LIN {X 0,Y 305.44,Z 814.433,A -85,B 0,C 180,E1 -16058.524,E2 -16058.524} C_VEL
LIN {X 0,Y 305.442,Z 814.432,A -85,B 0,C 180,E1 -16062.581,E2 -16062.581} C_VEL
LIN {X 0,Y 305.428,Z 814.435,A -85,B 0,C 180,E1 -16066.343,E2 -16066.343} C_VEL
LIN {X 0,Y 305.416,Z 814.438,A -85,B 0,C 180,E1 -16069.883,E2 -16069.883} C_VEL
LIN {X 0,Y 305.469,Z 814.43,A -85,B 0,C 180,E1 -16073.635,E2 -16073.635} C_VEL
LIN {X 0,Y 305.472,Z 814.433,A -85,B 0,C 180,E1 -16076.482,E2 -16076.482} C_VEL
LIN {X 0,Y 305.465,Z 814.429,A -85,B 0,C 180,E1 -16079.589,E2 -16079.589} C_VEL
LIN {X 0,Y 305.525,Z 814.42,A -85,B 0,C 180,E1 -16082.607,E2 -16082.607} C_VEL
LIN {X 0,Y 305.514,Z 814.416,A -85,B 0,C 180,E1 -16085.537,E2 -16085.537} C_VEL
LIN {X 0,Y 305.53,Z 814.621,A -85,B 0,C 180,E1 -16086.942,E2 -16086.942} C_VEL
LIN {X 0,Y 309.571,Z 825.379,A -85,B 0,C 180,E1 -16088.102,E2 -16088.102} C_VEL
LIN {X 0,Y 313.039,Z 835.887,A -85,B 0,C 180,E1 -16089.429,E2 -16089.429} C_VEL
LIN {X 0,Y 314.602,Z 841.496,A -85,B 0,C 180,E1 -16090.215,E2 -16090.215} C_VEL
LIN {X 0,Y 314.626,Z 844.023,A -85,B 0,C 180,E1 -16090.531,E2 -16090.531} C_VEL
LIN {X 0,Y 313.227,Z 855.02,A -85,B 0,C 180,E1 -16092.028,E2 -16092.028} C_VEL
LIN {X 0,Y 311.993,Z 864.467,A -85,B 0,C 180,E1 -16093.644,E2 -16093.644} C_VEL
LIN {X 0,Y 310.638,Z 872.23,A -85,B 0,C 180,E1 -16095.252,E2 -16095.252} C_VEL
LIN {X 0,Y 309.416,Z 879.778,A -85,B 0,C 180,E1 -16097.203,E2 -16097.203} C_VEL
LIN {X 0,Y 308.401,Z 886.662,A -85,B 0,C 180,E1 -16099.494,E2 -16099.494} C_VEL
LIN {X 0,Y 307.337,Z 891.297,A -85,B 0,C 180,E1 -16101.45,E2 -16101.45} C_VEL
LIN {X 0,Y 306.627,Z 894.819,A -85,B 0,C 180,E1 -16103.417,E2 -16103.417} C_VEL
LIN {X 0,Y 306.285,Z 896.636,A -85,B 0,C 180,E1 -16104.731,E2 -16104.731} C_VEL
LIN {X 0,Y 306.262,Z 897.968,A -85,B 0,C 180,E1 -16106.05,E2 -16106.05} C_VEL
LIN {X 0,Y 305.907,Z 899.547,A -85,B 0,C 180,E1 -16108.681,E2 -16108.681} C_VEL
LIN {X 0,Y 305.854,Z 899.777,A -85,B 0,C 180,E1 -16109.998,E2 -16109.998} C_VEL
LIN {X 0,Y 306.065,Z 899.011,A -85,B 0,C 180,E1 -16112.63,E2 -16112.63} C_VEL
LIN {X 0,Y 306.234,Z 898.069,A -85,B 0,C 180,E1 -16113.945,E2 -16113.945} C_VEL
LIN {X 0,Y 306.271,Z 896.777,A -85,B 0,C 180,E1 -16115.264,E2 -16115.264} C_VEL
LIN {X 0,Y 306.812,Z 893.971,A -85,B 0,C 180,E1 -16117.235,E2 -16117.235} C_VEL
LIN {X 0,Y 307.762,Z 890.128,A -85,B 0,C 180,E1 -16119.196,E2 -16119.196} C_VEL
LIN {X 0,Y 308.658,Z 885.217,A -85,B 0,C 180,E1 -16121.157,E2 -16121.157} C_VEL
LIN {X 0,Y 309.542,Z 879.05,A -85,B 0,C 180,E1 -16123.121,E2 -16123.121} C_VEL
LIN {X 0,Y 310.901,Z 871.272,A -85,B 0,C 180,E1 -16125.065,E2 -16125.065} C_VEL
LIN {X 0,Y 312.12,Z 863.342,A -85,B 0,C 180,E1 -16126.681,E2 -16126.681} C_VEL
LIN {X 0,Y 313.469,Z 853.646,A -85,B 0,C 180,E1 -16128.291,E2 -16128.291} C_VEL
LIN {X 0,Y 314.799,Z 842.532,A -85,B 0,C 180,E1 -16129.754,E2 -16129.754} C_VEL
LIN {X 0,Y 312.013,Z 832.57,A -85,B 0,C 180,E1 -16131.122,E2 -16131.122} C_VEL
LIN {X 0,Y 308.05,Z 821.176,A -85,B 0,C 180,E1 -16132.485,E2 -16132.485} C_VEL
LIN {X 0,Y 305.498,Z 814.43,A -85,B 0,C 180,E1 -16133.22,E2 -16133.22} C_VEL
LIN {X 0,Y 305.543,Z 814.427,A -85,B 0,C 180,E1 -16136.225,E2 -16136.225} C_VEL
LIN {X 0,Y 305.49,Z 814.432,A -85,B 0,C 180,E1 -16139.047,E2 -16139.047} C_VEL
LIN {X 0,Y 305.439,Z 814.44,A -85,B 0,C 180,E1 -16141.949,E2 -16141.949} C_VEL
LIN {X 0,Y 305.455,Z 814.436,A -85,B 0,C 180,E1 -16145.111,E2 -16145.111} C_VEL
LIN {X 0,Y 305.486,Z 814.434,A -85,B 0,C 180,E1 -16148.537,E2 -16148.537} C_VEL
LIN {X 0,Y 305.513,Z 814.43,A -85,B 0,C 180,E1 -16152.597,E2 -16152.597} C_VEL
LIN {X 0,Y 305.524,Z 814.427,A -85,B 0,C 180,E1 -16156.362,E2 -16156.362} C_VEL
LIN {X 0,Y 305.489,Z 814.431,A -85,B 0,C 180,E1 -16159.897,E2 -16159.897} C_VEL
LIN {X 0,Y 305.491,Z 814.43,A -85,B 0,C 180,E1 -16163.624,E2 -16163.624} C_VEL
LIN {X 0,Y 305.452,Z 814.432,A -85,B 0,C 180,E1 -16166.481,E2 -16166.481} C_VEL
LIN {X 0,Y 305.45,Z 814.429,A -85,B 0,C 180,E1 -16169.589,E2 -16169.589} C_VEL
LIN {X 0,Y 305.508,Z 814.431,A -85,B 0,C 180,E1 -16172.607,E2 -16172.607} C_VEL
LIN {X 0,Y 305.493,Z 814.428,A -85,B 0,C 180,E1 -16175.537,E2 -16175.537} C_VEL
LIN {X 0,Y 305.505,Z 814.424,A -85,B 0,C 180,E1 -16179.814,E2 -16179.814} C_VEL
LIN {X 0,Y 305.559,Z 814.423,A -85,B 0,C 180,E1 -16182.602,E2 -16182.602} C_VEL
LIN {X 0,Y 305.608,Z 814.407,A -85,B 0,C 180,E1 -16184.792,E2 -16184.792} C_VEL
LIN {X 0,Y 304.99,Z 814.49,A -85,B 0,C 180,E1 -16185.891,E2 -16185.891} C_VEL
LIN {X 0,Y 302.121,Z 814.853,A -85,B 0,C 180,E1 -16187.68,E2 -16187.68} C_VEL
LIN {X 0,Y 299.698,Z 815.153,A -85,B 0,C 180,E1 -16189.132,E2 -16189.132} C_VEL
LIN {X 0,Y 298.722,Z 815.27,A -85,B 0,C 180,E1 -16190.257,E2 -16190.257} C_VEL
LIN {X 0,Y 298.678,Z 815.274,A -85,B 0,C 180,E1 -16190.638,E2 -16190.638} C_VEL
LIN {X 0,Y 298.775,Z 815.272,A -85,B 0,C 180,E1 -16193.246,E2 -16193.246} C_VEL
LIN {X 0,Y 298.909,Z 815.252,A -85,B 0,C 180,E1 -16198.653,E2 -16198.653} C_VEL
LIN {X 0,Y 298.907,Z 815.256,A -85,B 0,C 180,E1 -16201.347,E2 -16201.347} C_VEL
LIN {X 0,Y 298.761,Z 815.268,A -85,B 0,C 180,E1 -16206.755,E2 -16206.755} C_VEL
LIN {X 0,Y 298.665,Z 815.282,A -85,B 0,C 180,E1 -16209.481,E2 -16209.481} C_VEL
LIN {X 0,Y 298.537,Z 815.294,A -85,B 0,C 180,E1 -16213.616,E2 -16213.616} C_VEL
LIN {X 0,Y 298.533,Z 815.3,A -85,B 0,C 180,E1 -16216.41,E2 -16216.41} C_VEL
LIN {X 0,Y 298.482,Z 815.307,A -85,B 0,C 180,E1 -16219.648,E2 -16219.648} C_VEL
LIN {X 0,Y 298.405,Z 815.315,A -85,B 0,C 180,E1 -16223.602,E2 -16223.602} C_VEL
LIN {X 0,Y 298.393,Z 815.314,A -85,B 0,C 180,E1 -16226.584,E2 -16226.584} C_VEL
LIN {X 0,Y 298.379,Z 815.318,A -85,B 0,C 180,E1 -16229.646,E2 -16229.646} C_VEL
LIN {X 0,Y 298.379,Z 815.315,A -85,B 0,C 180,E1 -16232.802,E2 -16232.802} C_VEL
LIN {X 0,Y 298.412,Z 815.313,A -85,B 0,C 180,E1 -16236.804,E2 -16236.804} C_VEL
LIN {X 0,Y 298.377,Z 815.387,A -85,B 0,C 180,E1 -16238.992,E2 -16238.992} C_VEL
LIN {X 0,Y 299.932,Z 822.588,A -85,B 0,C 180,E1 -16242.807,E2 -16242.807} C_VEL
LIN {X 0,Y 301.331,Z 829.707,A -85,B 0,C 180,E1 -16246.304,E2 -16246.304} C_VEL
LIN {X 0,Y 302.827,Z 837.684,A -85,B 0,C 180,E1 -16249.984,E2 -16249.984} C_VEL
LIN {X 0,Y 303.329,Z 842.26,A -85,B 0,C 180,E1 -16251.977,E2 -16251.977} C_VEL
LIN {X 0,Y 301.773,Z 852.318,A -85,B 0,C 180,E1 -16256.021,E2 -16256.021} C_VEL
LIN {X 0,Y 300.161,Z 863.757,A -85,B 0,C 180,E1 -16260.551,E2 -16260.551} C_VEL
LIN {X 0,Y 299.075,Z 873.062,A -85,B 0,C 180,E1 -16264.235,E2 -16264.235} C_VEL
LIN {X 0,Y 298.743,Z 875.947,A -85,B 0,C 180,E1 -16265.392,E2 -16265.392} C_VEL
LIN {X 0,Y 301.044,Z 890.754,A -85,B 0,C 180,E1 -16266.184,E2 -16266.184} C_VEL
LIN {X 0,Y 302.283,Z 903.528,A -85,B 0,C 180,E1 -16267.084,E2 -16267.084} C_VEL
LIN {X 0,Y 302.853,Z 916.115,A -85,B 0,C 180,E1 -16268.207,E2 -16268.207} C_VEL
LIN {X 0,Y 302.779,Z 927.553,A -85,B 0,C 180,E1 -16269.462,E2 -16269.462} C_VEL
LIN {X 0,Y 302.496,Z 939.049,A -85,B 0,C 180,E1 -16271.021,E2 -16271.021} C_VEL
LIN {X 0,Y 300.879,Z 949.163,A -85,B 0,C 180,E1 -16272.676,E2 -16272.676} C_VEL
LIN {X 0,Y 299.339,Z 957.948,A -85,B 0,C 180,E1 -16274.448,E2 -16274.448} C_VEL
LIN {X 0,Y 298.85,Z 963.193,A -85,B 0,C 180,E1 -16275.707,E2 -16275.707} C_VEL
LIN {X 0,Y 297.998,Z 970.299,A -85,B 0,C 180,E1 -16277.748,E2 -16277.748} C_VEL
LIN {X 0,Y 297.548,Z 976.039,A -85,B 0,C 180,E1 -16279.799,E2 -16279.799} C_VEL
LIN {X 0,Y 297.448,Z 980.589,A -85,B 0,C 180,E1 -16281.853,E2 -16281.853} C_VEL
LIN {X 0,Y 297.472,Z 983.012,A -85,B 0,C 180,E1 -16283.218,E2 -16283.218} C_VEL
LIN {X 0,Y 297.618,Z 984.994,A -85,B 0,C 180,E1 -16284.582,E2 -16284.582} C_VEL
LIN {X 0,Y 297.831,Z 986.496,A -85,B 0,C 180,E1 -16285.943,E2 -16285.943} C_VEL
LIN {X 0,Y 297.891,Z 987.553,A -85,B 0,C 180,E1 -16287.298,E2 -16287.298} C_VEL
LIN {X 0,Y 298.002,Z 988.207,A -85,B 0,C 180,E1 -16288.651,E2 -16288.651} C_VEL
LIN {X 0,Y 298.107,Z 988.446,A -85,B 0,C 180,E1 -16290.002,E2 -16290.002} C_VEL
LIN {X 0,Y 298.002,Z 988.199,A -85,B 0,C 180,E1 -16291.354,E2 -16291.354} C_VEL
LIN {X 0,Y 297.891,Z 987.539,A -85,B 0,C 180,E1 -16292.707,E2 -16292.707} C_VEL
LIN {X 0,Y 297.833,Z 986.476,A -85,B 0,C 180,E1 -16294.062,E2 -16294.062} C_VEL
LIN {X 0,Y 297.643,Z 984.969,A -85,B 0,C 180,E1 -16295.422,E2 -16295.422} C_VEL
LIN {X 0,Y 297.498,Z 982.359,A -85,B 0,C 180,E1 -16297.162,E2 -16297.162} C_VEL
LIN {X 0,Y 297.491,Z 977.661,A -85,B 0,C 180,E1 -16299.521,E2 -16299.521} C_VEL
LIN {X 0,Y 298.392,Z 967.682,A -85,B 0,C 180,E1 -16303.278,E2 -16303.278} C_VEL
LIN {X 0,Y 299.531,Z 960.67,A -85,B 0,C 180,E1 -16305.381,E2 -16305.381} C_VEL
LIN {X 0,Y 300.989,Z 952.878,A -85,B 0,C 180,E1 -16307.322,E2 -16307.322} C_VEL
LIN {X 0,Y 303.06,Z 943.402,A -85,B 0,C 180,E1 -16309.299,E2 -16309.299} C_VEL
LIN {X 0,Y 303.917,Z 937.917,A -85,B 0,C 180,E1 -16310.298,E2 -16310.298} C_VEL
LIN {X 0,Y 305.208,Z 926.074,A -85,B 0,C 180,E1 -16312.229,E2 -16312.229} C_VEL
LIN {X 0,Y 306.364,Z 915.772,A -85,B 0,C 180,E1 -16313.67,E2 -16313.67} C_VEL
LIN {X 0,Y 306.771,Z 906.337,A -85,B 0,C 180,E1 -16314.907,E2 -16314.907} C_VEL
LIN {X 0,Y 306.2,Z 894.123,A -85,B 0,C 180,E1 -16316.473,E2 -16316.473} C_VEL
LIN {X 0,Y 304.586,Z 880.151,A -85,B 0,C 180,E1 -16318.251,E2 -16318.251} C_VEL
LIN {X 0,Y 303.634,Z 873.796,A -85,B 0,C 180,E1 -16319.085,E2 -16319.085} C_VEL
LIN {X 0,Y 302.505,Z 869.23,A -85,B 0,C 180,E1 -16319.728,E2 -16319.728} C_VEL
LIN {X 0,Y 302.255,Z 867.254,A -85,B 0,C 180,E1 -16319.964,E2 -16319.964} C_VEL
LIN {X 0,Y 300.849,Z 862.102,A -85,B 0,C 180,E1 -16320.774,E2 -16320.774} C_VEL
LIN {X 0,Y 300.628,Z 859.665,A -85,B 0,C 180,E1 -16321.051,E2 -16321.051} C_VEL
LIN {X 0,Y 302.037,Z 850.294,A -85,B 0,C 180,E1 -16324.758,E2 -16324.758} C_VEL
LIN {X 0,Y 303.328,Z 842.197,A -85,B 0,C 180,E1 -16328.023,E2 -16328.023} C_VEL
LIN {X 0,Y 302.806,Z 837.637,A -85,B 0,C 180,E1 -16330.011,E2 -16330.011} C_VEL
LIN {X 0,Y 301.531,Z 830.902,A -85,B 0,C 180,E1 -16333.084,E2 -16333.084} C_VEL
LIN {X 0,Y 300.145,Z 823.831,A -85,B 0,C 180,E1 -16336.544,E2 -16336.544} C_VEL
LIN {X 0,Y 298.681,Z 816.741,A -85,B 0,C 180,E1 -16340.338,E2 -16340.338} C_VEL
LIN {X 0,Y 298.7,Z 816.569,A -85,B 0,C 180,E1 -16343.969,E2 -16343.969} C_VEL
LIN {X 0,Y 299.03,Z 817.445,A -85,B 0,C 180,E1 -16347.792,E2 -16347.792} C_VEL
LIN {X 0,Y 300.255,Z 819.262,A -85,B 0,C 180,E1 -16348.469,E2 -16348.469} C_VEL
LIN {X 0,Y 301.892,Z 820.565,A -85,B 0,C 180,E1 -16349.192,E2 -16349.192} C_VEL
LIN {X 0,Y 302.749,Z 822.767,A -85,B 0,C 180,E1 -16349.762,E2 -16349.762} C_VEL
LIN {X 0,Y 304.546,Z 825.104,A -85,B 0,C 180,E1 -16350.596,E2 -16350.596} C_VEL
LIN {X 0,Y 309.547,Z 834.229,A -85,B 0,C 180,E1 -16353.136,E2 -16353.136} C_VEL
LIN {X 0,Y 312.916,Z 842.356,A -85,B 0,C 180,E1 -16355.124,E2 -16355.124} C_VEL
LIN {X 0,Y 315.127,Z 849.686,A -85,B 0,C 180,E1 -16356.79,E2 -16356.79} C_VEL
LIN {X 0,Y 316.071,Z 854.161,A -85,B 0,C 180,E1 -16357.79,E2 -16357.79} C_VEL
LIN {X 0,Y 313.395,Z 865.579,A -85,B 0,C 180,E1 -16359.66,E2 -16359.66} C_VEL
LIN {X 0,Y 310.922,Z 874.802,A -85,B 0,C 180,E1 -16361.552,E2 -16361.552} C_VEL
LIN {X 0,Y 308.314,Z 883.257,A -85,B 0,C 180,E1 -16363.774,E2 -16363.774} C_VEL
LIN {X 0,Y 306.038,Z 889.85,A -85,B 0,C 180,E1 -16366.047,E2 -16366.047} C_VEL
LIN {X 0,Y 304.334,Z 894.277,A -85,B 0,C 180,E1 -16368.004,E2 -16368.004} C_VEL
LIN {X 0,Y 303.33,Z 896.625,A -85,B 0,C 180,E1 -16369.318,E2 -16369.318} C_VEL
LIN {X 0,Y 301.502,Z 899.889,A -85,B 0,C 180,E1 -16371.96,E2 -16371.96} C_VEL
LIN {X 0,Y 300.975,Z 900.956,A -85,B 0,C 180,E1 -16373.295,E2 -16373.295} C_VEL
LIN {X 0,Y 299.994,Z 901.745,A -85,B 0,C 180,E1 -16375.97,E2 -16375.97} C_VEL
LIN {X 0,Y 299.557,Z 901.573,A -85,B 0,C 180,E1 -16377.311,E2 -16377.311} C_VEL
LIN {X 0,Y 299.221,Z 900.976,A -85,B 0,C 180,E1 -16378.654,E2 -16378.654} C_VEL
LIN {X 0,Y 298.823,Z 899.932,A -85,B 0,C 180,E1 -16380,E2 -16380} C_VEL
LIN {X 0,Y 298.797,Z 898.519,A -85,B 0,C 180,E1 -16381.348,E2 -16381.348} C_VEL
LIN {X 0,Y 298.499,Z 894.353,A -85,B 0,C 180,E1 -16384.05,E2 -16384.05} C_VEL
LIN {X 0,Y 298.949,Z 889.992,A -85,B 0,C 180,E1 -16386.073,E2 -16386.073} C_VEL
LIN {X 0,Y 299.264,Z 885.539,A -85,B 0,C 180,E1 -16387.761,E2 -16387.761} C_VEL
LIN {X 0,Y 299.601,Z 880.204,A -85,B 0,C 180,E1 -16389.451,E2 -16389.451} C_VEL
LIN {X 0,Y 300.221,Z 872.425,A -85,B 0,C 180,E1 -16391.477,E2 -16391.477} C_VEL
LIN {X 0,Y 300.895,Z 864.513,A -85,B 0,C 180,E1 -16393.164,E2 -16393.164} C_VEL
LIN {X 0,Y 301.56,Z 856.156,A -85,B 0,C 180,E1 -16394.682,E2 -16394.682} C_VEL
LIN {X 0,Y 302.288,Z 847.42,A -85,B 0,C 180,E1 -16396.027,E2 -16396.027} C_VEL
LIN {X 0,Y 303.107,Z 837.178,A -85,B 0,C 180,E1 -16397.369,E2 -16397.369} C_VEL
LIN {X 0,Y 303.152,Z 833.974,A -85,B 0,C 180,E1 -16397.74,E2 -16397.74} C_VEL
LIN {X 0,Y 299.913,Z 821.316,A -85,B 0,C 180,E1 -16399.152,E2 -16399.152} C_VEL
LIN {X 0,Y 298.457,Z 815.303,A -85,B 0,C 180,E1 -16399.756,E2 -16399.756} C_VEL
LIN {X 0,Y 298.388,Z 815.314,A -85,B 0,C 180,E1 -16403.604,E2 -16403.604} C_VEL
LIN {X 0,Y 298.408,Z 815.303,A -85,B 0,C 180,E1 -16406.582,E2 -16406.582} C_VEL
LIN {X 0,Y 298.364,Z 815.317,A -85,B 0,C 180,E1 -16409.647,E2 -16409.647} C_VEL
LIN {X 0,Y 298.4,Z 815.301,A -85,B 0,C 180,E1 -16412.8,E2 -16412.8} C_VEL
LIN {X 0,Y 298.433,Z 815.303,A -85,B 0,C 180,E1 -16416.801,E2 -16416.801} C_VEL
LIN {X 0,Y 298.381,Z 815.313,A -85,B 0,C 180,E1 -16419.491,E2 -16419.491} C_VEL
LIN {X 0,Y 298.378,Z 815.313,A -85,B 0,C 180,E1 -16423.096,E2 -16423.096} C_VEL
LIN {X 0,Y 298.378,Z 815.314,A -85,B 0,C 180,E1 -16426.914,E2 -16426.914} C_VEL
LIN {X 0,Y 298.363,Z 815.318,A -85,B 0,C 180,E1 -16431.016,E2 -16431.016} C_VEL
LIN {X 0,Y 298.412,Z 815.311,A -85,B 0,C 180,E1 -16433.927,E2 -16433.927} C_VEL
LIN {X 0,Y 298.402,Z 815.311,A -85,B 0,C 180,E1 -16437.198,E2 -16437.198} C_VEL
LIN {X 0,Y 298.434,Z 815.303,A -85,B 0,C 180,E1 -16440.615,E2 -16440.615} C_VEL
LIN {X 0,Y 298.485,Z 815.297,A -85,B 0,C 180,E1 -16443.475,E2 -16443.475} C_VEL
LIN {X 0,Y 298.49,Z 815.293,A -85,B 0,C 180,E1 -16446.334,E2 -16446.334} C_VEL
LIN {X 0,Y 299.711,Z 818.793,A -85,B 0,C 180,E1 -16446.693,E2 -16446.693} C_VEL
LIN {X 0,Y 303.487,Z 828.792,A -85,B 0,C 180,E1 -16447.866,E2 -16447.866} C_VEL
LIN {X 0,Y 306.967,Z 839.762,A -85,B 0,C 180,E1 -16449.337,E2 -16449.337} C_VEL
LIN {X 0,Y 308.062,Z 844.182,A -85,B 0,C 180,E1 -16449.987,E2 -16449.987} C_VEL
LIN {X 0,Y 306.718,Z 855.004,A -85,B 0,C 180,E1 -16451.46,E2 -16451.46} C_VEL
LIN {X 0,Y 305.513,Z 863.76,A -85,B 0,C 180,E1 -16452.942,E2 -16452.942} C_VEL
LIN {X 0,Y 303.852,Z 873.263,A -85,B 0,C 180,E1 -16454.915,E2 -16454.915} C_VEL
LIN {X 0,Y 302.568,Z 880.812,A -85,B 0,C 180,E1 -16456.909,E2 -16456.909} C_VEL
LIN {X 0,Y 301.506,Z 887.694,A -85,B 0,C 180,E1 -16459.25,E2 -16459.25} C_VEL
LIN {X 0,Y 300.393,Z 892.329,A -85,B 0,C 180,E1 -16461.251,E2 -16461.251} C_VEL
LIN {X 0,Y 299.649,Z 895.852,A -85,B 0,C 180,E1 -16463.263,E2 -16463.263} C_VEL
LIN {X 0,Y 299.29,Z 897.668,A -85,B 0,C 180,E1 -16464.608,E2 -16464.608} C_VEL
LIN {X 0,Y 299.258,Z 898.999,A -85,B 0,C 180,E1 -16465.958,E2 -16465.958} C_VEL
LIN {X 0,Y 298.885,Z 900.579,A -85,B 0,C 180,E1 -16468.65,E2 -16468.65} C_VEL
LIN {X 0,Y 298.831,Z 900.809,A -85,B 0,C 180,E1 -16469.998,E2 -16469.998} C_VEL
LIN {X 0,Y 299.051,Z 900.041,A -85,B 0,C 180,E1 -16472.692,E2 -16472.692} C_VEL
LIN {X 0,Y 299.233,Z 899.099,A -85,B 0,C 180,E1 -16474.038,E2 -16474.038} C_VEL
LIN {X 0,Y 299.277,Z 897.808,A -85,B 0,C 180,E1 -16475.387,E2 -16475.387} C_VEL
LIN {X 0,Y 299.844,Z 895.001,A -85,B 0,C 180,E1 -16477.404,E2 -16477.404} C_VEL
LIN {X 0,Y 300.831,Z 891.158,A -85,B 0,C 180,E1 -16479.409,E2 -16479.409} C_VEL
LIN {X 0,Y 301.769,Z 886.247,A -85,B 0,C 180,E1 -16481.415,E2 -16481.415} C_VEL
LIN {X 0,Y 302.717,Z 880.077,A -85,B 0,C 180,E1 -16483.422,E2 -16483.422} C_VEL
LIN {X 0,Y 304.126,Z 872.3,A -85,B 0,C 180,E1 -16485.409,E2 -16485.409} C_VEL
LIN {X 0,Y 305.397,Z 864.37,A -85,B 0,C 180,E1 -16487.06,E2 -16487.06} C_VEL
LIN {X 0,Y 306.808,Z 854.674,A -85,B 0,C 180,E1 -16488.702,E2 -16488.702} C_VEL
LIN {X 0,Y 308.046,Z 843.929,A -85,B 0,C 180,E1 -16490.162,E2 -16490.162} C_VEL
LIN {X 0,Y 305.137,Z 833.647,A -85,B 0,C 180,E1 -16491.621,E2 -16491.621} C_VEL
LIN {X 0,Y 301.429,Z 823.117,A -85,B 0,C 180,E1 -16492.933,E2 -16492.933} C_VEL
LIN {X 0,Y 298.538,Z 815.657,A -85,B 0,C 180,E1 -16493.753,E2 -16493.753} C_VEL
LIN {X 0,Y 298.465,Z 815.308,A -85,B 0,C 180,E1 -16493.842,E2 -16493.842} C_VEL
LIN {X 0,Y 298.485,Z 815.305,A -85,B 0,C 180,E1 -16496.572,E2 -16496.572} C_VEL
LIN {X 0,Y 298.415,Z 815.314,A -85,B 0,C 180,E1 -16499.638,E2 -16499.638} C_VEL
LIN {X 0,Y 298.39,Z 815.317,A -85,B 0,C 180,E1 -16502.797,E2 -16502.797} C_VEL
LIN {X 0,Y 298.463,Z 815.308,A -85,B 0,C 180,E1 -16506.811,E2 -16506.811} C_VEL
LIN {X 0,Y 298.448,Z 815.307,A -85,B 0,C 180,E1 -16511.247,E2 -16511.247} C_VEL
LIN {X 0,Y 298.48,Z 815.304,A -85,B 0,C 180,E1 -16515.059,E2 -16515.059} C_VEL
LIN {X 0,Y 298.446,Z 815.309,A -85,B 0,C 180,E1 -16518.895,E2 -16518.895} C_VEL
LIN {X 0,Y 298.46,Z 815.306,A -85,B 0,C 180,E1 -16523.184,E2 -16523.184} C_VEL
LIN {X 0,Y 298.383,Z 815.316,A -85,B 0,C 180,E1 -16527.198,E2 -16527.198} C_VEL
LIN {X 0,Y 298.419,Z 815.307,A -85,B 0,C 180,E1 -16530.613,E2 -16530.613} C_VEL
LIN {X 0,Y 298.47,Z 815.301,A -85,B 0,C 180,E1 -16533.473,E2 -16533.473} C_VEL
LIN {X 0,Y 298.421,Z 815.313,A -85,B 0,C 180,E1 -16536.696,E2 -16536.696} C_VEL
LIN {X 0,Y 298.524,Z 815.297,A -85,B 0,C 180,E1 -16540.756,E2 -16540.756} C_VEL
LIN {X 0,Y 298.578,Z 815.284,A -85,B 0,C 180,E1 -16544.994,E2 -16544.994} C_VEL
LIN {X 0,Y 298.58,Z 815.293,A -85,B 0,C 180,E1 -16549.146,E2 -16549.146} C_VEL
LIN {X 0,Y 298.678,Z 815.274,A -85,B 0,C 180,E1 -16550.638,E2 -16550.638} C_VEL
LIN {X 0,Y 298.068,Z 815.354,A -85,B 0,C 180,E1 -16551.764,E2 -16551.764} C_VEL
LIN {X 0,Y 295.121,Z 815.729,A -85,B 0,C 180,E1 -16553.595,E2 -16553.595} C_VEL
LIN {X 0,Y 292.639,Z 816.037,A -85,B 0,C 180,E1 -16555.082,E2 -16555.082} C_VEL
LIN {X 0,Y 291.67,Z 816.148,A -85,B 0,C 180,E1 -16556.236,E2 -16556.236} C_VEL
LIN {X 0,Y 291.647,Z 816.149,A -85,B 0,C 180,E1 -16556.627,E2 -16556.627} C_VEL
LIN {X 0,Y 291.949,Z 816.122,A -85,B 0,C 180,E1 -16560,E2 -16560} C_VEL
LIN {X 0,Y 291.771,Z 816.143,A -85,B 0,C 180,E1 -16562.761,E2 -16562.761} C_VEL
LIN {X 0,Y 291.712,Z 816.146,A -85,B 0,C 180,E1 -16566.919,E2 -16566.919} C_VEL
LIN {X 0,Y 291.614,Z 816.162,A -85,B 0,C 180,E1 -16569.712,E2 -16569.712} C_VEL
LIN {X 0,Y 291.507,Z 816.173,A -85,B 0,C 180,E1 -16573.951,E2 -16573.951} C_VEL
LIN {X 0,Y 291.47,Z 816.179,A -85,B 0,C 180,E1 -16576.819,E2 -16576.819} C_VEL
LIN {X 0,Y 291.436,Z 816.185,A -85,B 0,C 180,E1 -16579.876,E2 -16579.876} C_VEL
LIN {X 0,Y 291.345,Z 816.196,A -85,B 0,C 180,E1 -16584.21,E2 -16584.21} C_VEL
LIN {X 0,Y 291.339,Z 816.19,A -85,B 0,C 180,E1 -16587.28,E2 -16587.28} C_VEL
LIN {X 0,Y 291.304,Z 816.196,A -85,B 0,C 180,E1 -16590.441,E2 -16590.441} C_VEL
LIN {X 0,Y 291.329,Z 816.196,A -85,B 0,C 180,E1 -16593.7,E2 -16593.7} C_VEL
LIN {X 0,Y 291.34,Z 816.195,A -85,B 0,C 180,E1 -16597.25,E2 -16597.25} C_VEL
LIN {X 0,Y 291.373,Z 816.376,A -85,B 0,C 180,E1 -16598.408,E2 -16598.408} C_VEL
LIN {X 0,Y 292.831,Z 823.332,A -85,B 0,C 180,E1 -16602.222,E2 -16602.222} C_VEL
LIN {X 0,Y 294.255,Z 830.291,A -85,B 0,C 180,E1 -16605.768,E2 -16605.768} C_VEL
LIN {X 0,Y 295.702,Z 838.148,A -85,B 0,C 180,E1 -16609.513,E2 -16609.513} C_VEL
LIN {X 0,Y 296.331,Z 842.549,A -85,B 0,C 180,E1 -16611.504,E2 -16611.504} C_VEL
LIN {X 0,Y 295.439,Z 848.491,A -85,B 0,C 180,E1 -16613.979,E2 -16613.979} C_VEL
LIN {X 0,Y 294.404,Z 855.109,A -85,B 0,C 180,E1 -16616.701,E2 -16616.701} C_VEL
LIN {X 0,Y 292.809,Z 866.427,A -85,B 0,C 180,E1 -16621.315,E2 -16621.315} C_VEL
LIN {X 0,Y 291.843,Z 874.87,A -85,B 0,C 180,E1 -16624.77,E2 -16624.77} C_VEL
LIN {X 0,Y 294.112,Z 889.571,A -85,B 0,C 180,E1 -16625.582,E2 -16625.582} C_VEL
LIN {X 0,Y 295.354,Z 901.517,A -85,B 0,C 180,E1 -16626.444,E2 -16626.444} C_VEL
LIN {X 0,Y 295.953,Z 913.283,A -85,B 0,C 180,E1 -16627.496,E2 -16627.496} C_VEL
LIN {X 0,Y 295.946,Z 925.435,A -85,B 0,C 180,E1 -16628.836,E2 -16628.836} C_VEL
LIN {X 0,Y 295.625,Z 936.804,A -85,B 0,C 180,E1 -16630.382,E2 -16630.382} C_VEL
LIN {X 0,Y 295.256,Z 941.268,A -85,B 0,C 180,E1 -16631.079,E2 -16631.079} C_VEL
LIN {X 0,Y 293.786,Z 949.936,A -85,B 0,C 180,E1 -16632.604,E2 -16632.604} C_VEL
LIN {X 0,Y 292.307,Z 957.749,A -85,B 0,C 180,E1 -16634.264,E2 -16634.264} C_VEL
LIN {X 0,Y 291.519,Z 964.677,A -85,B 0,C 180,E1 -16636.052,E2 -16636.052} C_VEL
LIN {X 0,Y 290.767,Z 971.326,A -85,B 0,C 180,E1 -16638.147,E2 -16638.147} C_VEL
LIN {X 0,Y 290.443,Z 976.657,A -85,B 0,C 180,E1 -16640.251,E2 -16640.251} C_VEL
LIN {X 0,Y 290.384,Z 981.698,A -85,B 0,C 180,E1 -16642.886,E2 -16642.886} C_VEL
LIN {X 0,Y 290.535,Z 983.95,A -85,B 0,C 180,E1 -16644.45,E2 -16644.45} C_VEL
LIN {X 0,Y 290.784,Z 985.459,A -85,B 0,C 180,E1 -16645.845,E2 -16645.845} C_VEL
LIN {X 0,Y 290.848,Z 986.518,A -85,B 0,C 180,E1 -16647.232,E2 -16647.232} C_VEL
LIN {X 0,Y 290.966,Z 987.174,A -85,B 0,C 180,E1 -16648.618,E2 -16648.618} C_VEL
LIN {X 0,Y 291.079,Z 987.414,A -85,B 0,C 180,E1 -16650.002,E2 -16650.002} C_VEL
LIN {X 0,Y 290.966,Z 987.166,A -85,B 0,C 180,E1 -16651.387,E2 -16651.387} C_VEL
LIN {X 0,Y 290.849,Z 986.503,A -85,B 0,C 180,E1 -16652.772,E2 -16652.772} C_VEL
LIN {X 0,Y 290.788,Z 985.439,A -85,B 0,C 180,E1 -16654.16,E2 -16654.16} C_VEL
LIN {X 0,Y 290.563,Z 983.925,A -85,B 0,C 180,E1 -16655.554,E2 -16655.554} C_VEL
LIN {X 0,Y 290.398,Z 980.8,A -85,B 0,C 180,E1 -16657.651,E2 -16657.651} C_VEL
LIN {X 0,Y 290.451,Z 976.612,A -85,B 0,C 180,E1 -16659.754,E2 -16659.754} C_VEL
LIN {X 0,Y 291.015,Z 970.065,A -85,B 0,C 180,E1 -16662.556,E2 -16662.556} C_VEL
LIN {X 0,Y 291.96,Z 964.021,A -85,B 0,C 180,E1 -16664.643,E2 -16664.643} C_VEL
LIN {X 0,Y 293.083,Z 957.966,A -85,B 0,C 180,E1 -16666.426,E2 -16666.426} C_VEL
LIN {X 0,Y 294.479,Z 951.424,A -85,B 0,C 180,E1 -16668.077,E2 -16668.077} C_VEL
LIN {X 0,Y 296.808,Z 942.004,A -85,B 0,C 180,E1 -16670.083,E2 -16670.083} C_VEL
LIN {X 0,Y 297.97,Z 932.674,A -85,B 0,C 180,E1 -16671.809,E2 -16671.809} C_VEL
LIN {X 0,Y 299.448,Z 922.056,A -85,B 0,C 180,E1 -16673.517,E2 -16673.517} C_VEL
LIN {X 0,Y 300.488,Z 912.384,A -85,B 0,C 180,E1 -16674.9,E2 -16674.9} C_VEL
LIN {X 0,Y 300.654,Z 902.867,A -85,B 0,C 180,E1 -16676.226,E2 -16676.226} C_VEL
LIN {X 0,Y 299.979,Z 890.384,A -85,B 0,C 180,E1 -16677.943,E2 -16677.943} C_VEL
LIN {X 0,Y 298.6,Z 878.323,A -85,B 0,C 180,E1 -16679.624,E2 -16679.624} C_VEL
LIN {X 0,Y 297.247,Z 870.25,A -85,B 0,C 180,E1 -16680.831,E2 -16680.831} C_VEL
LIN {X 0,Y 295.517,Z 862.218,A -85,B 0,C 180,E1 -16682.105,E2 -16682.105} C_VEL
LIN {X 0,Y 294.444,Z 857.057,A -85,B 0,C 180,E1 -16682.967,E2 -16682.967} C_VEL
LIN {X 0,Y 294.346,Z 855.281,A -85,B 0,C 180,E1 -16683.208,E2 -16683.208} C_VEL
LIN {X 0,Y 296.022,Z 845.418,A -85,B 0,C 180,E1 -16687.261,E2 -16687.261} C_VEL
LIN {X 0,Y 296.321,Z 842.495,A -85,B 0,C 180,E1 -16688.493,E2 -16688.493} C_VEL
LIN {X 0,Y 295.2,Z 835.25,A -85,B 0,C 180,E1 -16691.809,E2 -16691.809} C_VEL
LIN {X 0,Y 293.501,Z 826.652,A -85,B 0,C 180,E1 -16696.019,E2 -16696.019} C_VEL
LIN {X 0,Y 292.503,Z 821.725,A -85,B 0,C 180,E1 -16698.671,E2 -16698.671} C_VEL
LIN {X 0,Y 292.81,Z 820.89,A -85,B 0,C 180,E1 -16700.183,E2 -16700.183} C_VEL
LIN {X 0,Y 292.765,Z 820.404,A -85,B 0,C 180,E1 -16703.12,E2 -16703.12} C_VEL
LIN {X 0,Y 292.887,Z 820.749,A -85,B 0,C 180,E1 -16705.601,E2 -16705.601} C_VEL
LIN {X 0,Y 296.238,Z 824.189,A -85,B 0,C 180,E1 -16707.636,E2 -16707.636} C_VEL
LIN {X 0,Y 298.344,Z 826.505,A -85,B 0,C 180,E1 -16708.785,E2 -16708.785} C_VEL
LIN {X 0,Y 300.301,Z 830.315,A -85,B 0,C 180,E1 -16709.991,E2 -16709.991} C_VEL
LIN {X 0,Y 303.313,Z 835.614,A -85,B 0,C 180,E1 -16711.705,E2 -16711.705} C_VEL
LIN {X 0,Y 306.771,Z 843.679,A -85,B 0,C 180,E1 -16713.911,E2 -16713.911} C_VEL
LIN {X 0,Y 309.413,Z 852.423,A -85,B 0,C 180,E1 -16716.101,E2 -16716.101} C_VEL
LIN {X 0,Y 310.331,Z 856.898,A -85,B 0,C 180,E1 -16717.162,E2 -16717.162} C_VEL
LIN {X 0,Y 307.747,Z 867.133,A -85,B 0,C 180,E1 -16718.919,E2 -16718.919} C_VEL
LIN {X 0,Y 305.172,Z 876.002,A -85,B 0,C 180,E1 -16720.777,E2 -16720.777} C_VEL
LIN {X 0,Y 302.606,Z 883.48,A -85,B 0,C 180,E1 -16722.755,E2 -16722.755} C_VEL
LIN {X 0,Y 300.201,Z 890.395,A -85,B 0,C 180,E1 -16725.077,E2 -16725.077} C_VEL
LIN {X 0,Y 297.677,Z 896.226,A -85,B 0,C 180,E1 -16727.732,E2 -16727.732} C_VEL
LIN {X 0,Y 296.6,Z 898.411,A -85,B 0,C 180,E1 -16729.073,E2 -16729.073} C_VEL
LIN {X 0,Y 295.595,Z 900.144,A -85,B 0,C 180,E1 -16730.42,E2 -16730.42} C_VEL
LIN {X 0,Y 294.653,Z 901.458,A -85,B 0,C 180,E1 -16731.772,E2 -16731.772} C_VEL
LIN {X 0,Y 294.081,Z 902.418,A -85,B 0,C 180,E1 -16733.137,E2 -16733.137} C_VEL
LIN {X 0,Y 293.041,Z 903.028,A -85,B 0,C 180,E1 -16735.874,E2 -16735.874} C_VEL
LIN {X 0,Y 292.577,Z 902.752,A -85,B 0,C 180,E1 -16737.246,E2 -16737.246} C_VEL
LIN {X 0,Y 292.217,Z 902.034,A -85,B 0,C 180,E1 -16738.622,E2 -16738.622} C_VEL
LIN {X 0,Y 291.773,Z 899.419,A -85,B 0,C 180,E1 -16741.38,E2 -16741.38} C_VEL
LIN {X 0,Y 291.547,Z 896.334,A -85,B 0,C 180,E1 -16743.455,E2 -16743.455} C_VEL
LIN {X 0,Y 291.719,Z 892.198,A -85,B 0,C 180,E1 -16745.53,E2 -16745.53} C_VEL
LIN {X 0,Y 292.228,Z 885.865,A -85,B 0,C 180,E1 -16747.949,E2 -16747.949} C_VEL
LIN {X 0,Y 292.579,Z 880.355,A -85,B 0,C 180,E1 -16749.68,E2 -16749.68} C_VEL
LIN {X 0,Y 293.247,Z 872.432,A -85,B 0,C 180,E1 -16751.754,E2 -16751.754} C_VEL
LIN {X 0,Y 293.936,Z 864.268,A -85,B 0,C 180,E1 -16753.481,E2 -16753.481} C_VEL
LIN {X 0,Y 294.552,Z 856.707,A -85,B 0,C 180,E1 -16754.862,E2 -16754.862} C_VEL
LIN {X 0,Y 295.305,Z 847.884,A -85,B 0,C 180,E1 -16756.239,E2 -16756.239} C_VEL
LIN {X 0,Y 296.112,Z 837.696,A -85,B 0,C 180,E1 -16757.593,E2 -16757.593} C_VEL
LIN {X 0,Y 295.977,Z 834.492,A -85,B 0,C 180,E1 -16757.98,E2 -16757.98} C_VEL
LIN {X 0,Y 292.955,Z 822.593,A -85,B 0,C 180,E1 -16759.334,E2 -16759.334} C_VEL
LIN {X 0,Y 291.396,Z 816.18,A -85,B 0,C 180,E1 -16759.974,E2 -16759.974} C_VEL
LIN {X 0,Y 291.332,Z 816.194,A -85,B 0,C 180,E1 -16764.211,E2 -16764.211} C_VEL
LIN {X 0,Y 291.335,Z 816.183,A -85,B 0,C 180,E1 -16767.281,E2 -16767.281} C_VEL
LIN {X 0,Y 291.309,Z 816.194,A -85,B 0,C 180,E1 -16770.44,E2 -16770.44} C_VEL
LIN {X 0,Y 291.351,Z 816.183,A -85,B 0,C 180,E1 -16773.698,E2 -16773.698} C_VEL
LIN {X 0,Y 291.359,Z 816.184,A -85,B 0,C 180,E1 -16777.247,E2 -16777.247} C_VEL
LIN {X 0,Y 291.307,Z 816.195,A -85,B 0,C 180,E1 -16780.647,E2 -16780.647} C_VEL
LIN {X 0,Y 291.289,Z 816.201,A -85,B 0,C 180,E1 -16784.402,E2 -16784.402} C_VEL
LIN {X 0,Y 291.302,Z 816.199,A -85,B 0,C 180,E1 -16788.41,E2 -16788.41} C_VEL
LIN {X 0,Y 291.394,Z 816.182,A -85,B 0,C 180,E1 -16792.915,E2 -16792.915} C_VEL
LIN {X 0,Y 291.351,Z 816.193,A -85,B 0,C 180,E1 -16796.3,E2 -16796.3} C_VEL
LIN {X 0,Y 291.39,Z 816.183,A -85,B 0,C 180,E1 -16800.26,E2 -16800.26} C_VEL
LIN {X 0,Y 291.421,Z 816.179,A -85,B 0,C 180,E1 -16804.27,E2 -16804.27} C_VEL
LIN {X 0,Y 291.444,Z 816.168,A -85,B 0,C 180,E1 -16805.702,E2 -16805.702} C_VEL
LIN {X 0,Y 293.046,Z 820.65,A -85,B 0,C 180,E1 -16806.188,E2 -16806.188} C_VEL
LIN {X 0,Y 296.857,Z 830.606,A -85,B 0,C 180,E1 -16807.416,E2 -16807.416} C_VEL
LIN {X 0,Y 300.146,Z 841.111,A -85,B 0,C 180,E1 -16808.877,E2 -16808.877} C_VEL
LIN {X 0,Y 301.265,Z 845.251,A -85,B 0,C 180,E1 -16809.515,E2 -16809.515} C_VEL
LIN {X 0,Y 300.893,Z 849.934,A -85,B 0,C 180,E1 -16810.142,E2 -16810.142} C_VEL
LIN {X 0,Y 299.611,Z 859.181,A -85,B 0,C 180,E1 -16811.536,E2 -16811.536} C_VEL
LIN {X 0,Y 298.263,Z 868.206,A -85,B 0,C 180,E1 -16813.221,E2 -16813.221} C_VEL
LIN {X 0,Y 296.602,Z 876.984,A -85,B 0,C 180,E1 -16815.241,E2 -16815.241} C_VEL
LIN {X 0,Y 295.437,Z 883.882,A -85,B 0,C 180,E1 -16817.247,E2 -16817.247} C_VEL
LIN {X 0,Y 294.616,Z 888.725,A -85,B 0,C 180,E1 -16818.996,E2 -16818.996} C_VEL
LIN {X 0,Y 293.453,Z 893.362,A -85,B 0,C 180,E1 -16821.042,E2 -16821.042} C_VEL
LIN {X 0,Y 292.674,Z 896.884,A -85,B 0,C 180,E1 -16823.102,E2 -16823.102} C_VEL
LIN {X 0,Y 292.298,Z 898.7,A -85,B 0,C 180,E1 -16824.479,E2 -16824.479} C_VEL
LIN {X 0,Y 292.254,Z 900.03,A -85,B 0,C 180,E1 -16825.861,E2 -16825.861} C_VEL
LIN {X 0,Y 291.863,Z 901.61,A -85,B 0,C 180,E1 -16828.618,E2 -16828.618} C_VEL
LIN {X 0,Y 291.807,Z 901.84,A -85,B 0,C 180,E1 -16829.998,E2 -16829.998} C_VEL
LIN {X 0,Y 292.037,Z 901.072,A -85,B 0,C 180,E1 -16832.756,E2 -16832.756} C_VEL
LIN {X 0,Y 292.232,Z 900.129,A -85,B 0,C 180,E1 -16834.135,E2 -16834.135} C_VEL
LIN {X 0,Y 292.283,Z 898.838,A -85,B 0,C 180,E1 -16835.517,E2 -16835.517} C_VEL
LIN {X 0,Y 292.879,Z 896.032,A -85,B 0,C 180,E1 -16837.581,E2 -16837.581} C_VEL
LIN {X 0,Y 293.904,Z 892.188,A -85,B 0,C 180,E1 -16839.633,E2 -16839.633} C_VEL
LIN {X 0,Y 294.885,Z 887.276,A -85,B 0,C 180,E1 -16841.685,E2 -16841.685} C_VEL
LIN {X 0,Y 295.91,Z 881.103,A -85,B 0,C 180,E1 -16843.737,E2 -16843.737} C_VEL
LIN {X 0,Y 297.362,Z 873.328,A -85,B 0,C 180,E1 -16845.768,E2 -16845.768} C_VEL
LIN {X 0,Y 298.688,Z 865.398,A -85,B 0,C 180,E1 -16847.455,E2 -16847.455} C_VEL
LIN {X 0,Y 300.162,Z 855.702,A -85,B 0,C 180,E1 -16849.132,E2 -16849.132} C_VEL
LIN {X 0,Y 301.459,Z 846.137,A -85,B 0,C 180,E1 -16850.466,E2 -16850.466} C_VEL
LIN {X 0,Y 299.098,Z 837.399,A -85,B 0,C 180,E1 -16851.777,E2 -16851.777} C_VEL
LIN {X 0,Y 295.297,Z 826.229,A -85,B 0,C 180,E1 -16853.258,E2 -16853.258} C_VEL
LIN {X 0,Y 291.496,Z 816.555,A -85,B 0,C 180,E1 -16854.378,E2 -16854.378} C_VEL
LIN {X 0,Y 291.443,Z 816.182,A -85,B 0,C 180,E1 -16854.435,E2 -16854.435} C_VEL
LIN {X 0,Y 291.418,Z 816.185,A -85,B 0,C 180,E1 -16857.269,E2 -16857.269} C_VEL
LIN {X 0,Y 291.332,Z 816.196,A -85,B 0,C 180,E1 -16860.434,E2 -16860.434} C_VEL
LIN {X 0,Y 291.338,Z 816.196,A -85,B 0,C 180,E1 -16863.696,E2 -16863.696} C_VEL
LIN {X 0,Y 291.397,Z 816.188,A -85,B 0,C 180,E1 -16867.259,E2 -16867.259} C_VEL
LIN {X 0,Y 291.398,Z 816.188,A -85,B 0,C 180,E1 -16870.627,E2 -16870.627} C_VEL
LIN {X 0,Y 291.398,Z 816.189,A -85,B 0,C 180,E1 -16874.377,E2 -16874.377} C_VEL
LIN {X 0,Y 291.38,Z 816.187,A -85,B 0,C 180,E1 -16878.388,E2 -16878.388} C_VEL
LIN {X 0,Y 291.378,Z 816.182,A -85,B 0,C 180,E1 -16881.162,E2 -16881.162} C_VEL
LIN {X 0,Y 291.374,Z 816.186,A -85,B 0,C 180,E1 -16884.628,E2 -16884.628} C_VEL
LIN {X 0,Y 291.359,Z 816.19,A -85,B 0,C 180,E1 -16887.949,E2 -16887.949} C_VEL
LIN {X 0,Y 291.369,Z 816.19,A -85,B 0,C 180,E1 -16891.157,E2 -16891.157} C_VEL
LIN {X 0,Y 291.403,Z 816.182,A -85,B 0,C 180,E1 -16894.27,E2 -16894.27} C_VEL
LIN {X 0,Y 291.367,Z 816.19,A -85,B 0,C 180,E1 -16897.298,E2 -16897.298} C_VEL
LIN {X 0,Y 291.443,Z 816.176,A -85,B 0,C 180,E1 -16900.269,E2 -16900.269} C_VEL
LIN {X 0,Y 291.54,Z 816.16,A -85,B 0,C 180,E1 -16904.623,E2 -16904.623} C_VEL
LIN {X 0,Y 291.523,Z 816.174,A -85,B 0,C 180,E1 -16908.88,E2 -16908.88} C_VEL
LIN {X 0,Y 291.69,Z 816.147,A -85,B 0,C 180,E1 -16911.688,E2 -16911.688} C_VEL
LIN {X 0,Y 291.612,Z 816.163,A -85,B 0,C 180,E1 -16914.468,E2 -16914.468} C_VEL
LIN {X 0,Y 291.647,Z 816.149,A -85,B 0,C 180,E1 -16916.627,E2 -16916.627} C_VEL
LIN {X 0,Y 291.448,Z 816.177,A -85,B 0,C 180,E1 -16917.398,E2 -16917.398} C_VEL
LIN {X 0,Y 290.2,Z 816.34,A -85,B 0,C 180,E1 -16918.539,E2 -16918.539} C_VEL
LIN {X 0,Y 285.894,Z 816.877,A -85,B 0,C 180,E1 -16921.19,E2 -16921.19} C_VEL
LIN {X 0,Y 284.819,Z 817.009,A -85,B 0,C 180,E1 -16922.373,E2 -16922.373} C_VEL
LIN {X 0,Y 284.726,Z 817.021,A -85,B 0,C 180,E1 -16922.775,E2 -16922.775} C_VEL
LIN {X 0,Y 284.667,Z 817.025,A -85,B 0,C 180,E1 -16927.091,E2 -16927.091} C_VEL
LIN {X 0,Y 284.551,Z 817.042,A -85,B 0,C 180,E1 -16929.956,E2 -16929.956} C_VEL
LIN {X 0,Y 284.466,Z 817.052,A -85,B 0,C 180,E1 -16934.304,E2 -16934.304} C_VEL
LIN {X 0,Y 284.407,Z 817.059,A -85,B 0,C 180,E1 -16937.249,E2 -16937.249} C_VEL
LIN {X 0,Y 284.362,Z 817.067,A -85,B 0,C 180,E1 -16940.243,E2 -16940.243} C_VEL
LIN {X 0,Y 284.306,Z 817.072,A -85,B 0,C 180,E1 -16943.854,E2 -16943.854} C_VEL
LIN {X 0,Y 284.269,Z 817.072,A -85,B 0,C 180,E1 -16948.017,E2 -16948.017} C_VEL
LIN {X 0,Y 284.271,Z 817.075,A -85,B 0,C 180,E1 -16951.277,E2 -16951.277} C_VEL
LIN {X 0,Y 284.323,Z 817.068,A -85,B 0,C 180,E1 -16955.348,E2 -16955.348} C_VEL
LIN {X 0,Y 284.309,Z 817.218,A -85,B 0,C 180,E1 -16957.724,E2 -16957.724} C_VEL
LIN {X 0,Y 285.775,Z 824.049,A -85,B 0,C 180,E1 -16961.606,E2 -16961.606} C_VEL
LIN {X 0,Y 287.166,Z 830.872,A -85,B 0,C 180,E1 -16965.214,E2 -16965.214} C_VEL
LIN {X 0,Y 288.606,Z 838.602,A -85,B 0,C 180,E1 -16969.017,E2 -16969.017} C_VEL
LIN {X 0,Y 289.298,Z 842.873,A -85,B 0,C 180,E1 -16971.022,E2 -16971.022} C_VEL
LIN {X 0,Y 289.028,Z 846.382,A -85,B 0,C 180,E1 -16972.566,E2 -16972.566} C_VEL
LIN {X 0,Y 287.542,Z 854.961,A -85,B 0,C 180,E1 -16976.203,E2 -16976.203} C_VEL
LIN {X 0,Y 285.962,Z 865.345,A -85,B 0,C 180,E1 -16980.562,E2 -16980.562} C_VEL
LIN {X 0,Y 284.902,Z 873.763,A -85,B 0,C 180,E1 -16984.11,E2 -16984.11} C_VEL
LIN {X 0,Y 287.254,Z 888.672,A -85,B 0,C 180,E1 -16984.97,E2 -16984.97} C_VEL
LIN {X 0,Y 288.585,Z 901.612,A -85,B 0,C 180,E1 -16985.951,E2 -16985.951} C_VEL
LIN {X 0,Y 289.164,Z 913.953,A -85,B 0,C 180,E1 -16987.119,E2 -16987.119} C_VEL
LIN {X 0,Y 289.091,Z 925.731,A -85,B 0,C 180,E1 -16988.483,E2 -16988.483} C_VEL
LIN {X 0,Y 288.665,Z 936.902,A -85,B 0,C 180,E1 -16990.074,E2 -16990.074} C_VEL
LIN {X 0,Y 288.327,Z 941.282,A -85,B 0,C 180,E1 -16990.791,E2 -16990.791} C_VEL
LIN {X 0,Y 286.673,Z 950.6,A -85,B 0,C 180,E1 -16992.526,E2 -16992.526} C_VEL
LIN {X 0,Y 285.193,Z 958.31,A -85,B 0,C 180,E1 -16994.275,E2 -16994.275} C_VEL
LIN {X 0,Y 284.425,Z 964.828,A -85,B 0,C 180,E1 -16996.062,E2 -16996.062} C_VEL
LIN {X 0,Y 283.598,Z 972.17,A -85,B 0,C 180,E1 -16998.568,E2 -16998.568} C_VEL
LIN {X 0,Y 283.331,Z 977.11,A -85,B 0,C 180,E1 -17000.724,E2 -17000.724} C_VEL
LIN {X 0,Y 283.346,Z 980.925,A -85,B 0,C 180,E1 -17002.879,E2 -17002.879} C_VEL
LIN {X 0,Y 283.454,Z 982.906,A -85,B 0,C 180,E1 -17004.311,E2 -17004.311} C_VEL
LIN {X 0,Y 283.715,Z 984.419,A -85,B 0,C 180,E1 -17005.741,E2 -17005.741} C_VEL
LIN {X 0,Y 283.804,Z 985.483,A -85,B 0,C 180,E1 -17007.164,E2 -17007.164} C_VEL
LIN {X 0,Y 283.929,Z 986.141,A -85,B 0,C 180,E1 -17008.584,E2 -17008.584} C_VEL
LIN {X 0,Y 284.052,Z 986.382,A -85,B 0,C 180,E1 -17010.003,E2 -17010.003} C_VEL
LIN {X 0,Y 283.929,Z 986.132,A -85,B 0,C 180,E1 -17011.421,E2 -17011.421} C_VEL
LIN {X 0,Y 283.805,Z 985.468,A -85,B 0,C 180,E1 -17012.841,E2 -17012.841} C_VEL
LIN {X 0,Y 283.721,Z 984.398,A -85,B 0,C 180,E1 -17014.264,E2 -17014.264} C_VEL
LIN {X 0,Y 283.486,Z 982.88,A -85,B 0,C 180,E1 -17015.694,E2 -17015.694} C_VEL
LIN {X 0,Y 283.329,Z 979.752,A -85,B 0,C 180,E1 -17017.843,E2 -17017.843} C_VEL
LIN {X 0,Y 283.775,Z 971.182,A -85,B 0,C 180,E1 -17022.155,E2 -17022.155} C_VEL
LIN {X 0,Y 284.806,Z 964.759,A -85,B 0,C 180,E1 -17024.654,E2 -17024.654} C_VEL
LIN {X 0,Y 286.111,Z 958.446,A -85,B 0,C 180,E1 -17026.666,E2 -17026.666} C_VEL
LIN {X 0,Y 288.08,Z 950.075,A -85,B 0,C 180,E1 -17028.862,E2 -17028.862} C_VEL
LIN {X 0,Y 290.141,Z 942.396,A -85,B 0,C 180,E1 -17030.565,E2 -17030.565} C_VEL
LIN {X 0,Y 291.43,Z 933.542,A -85,B 0,C 180,E1 -17032.325,E2 -17032.325} C_VEL
LIN {X 0,Y 293.08,Z 923.409,A -85,B 0,C 180,E1 -17034.06,E2 -17034.06} C_VEL
LIN {X 0,Y 294.306,Z 914.32,A -85,B 0,C 180,E1 -17035.46,E2 -17035.46} C_VEL
LIN {X 0,Y 294.728,Z 902.425,A -85,B 0,C 180,E1 -17037.234,E2 -17037.234} C_VEL
LIN {X 0,Y 294.288,Z 890.792,A -85,B 0,C 180,E1 -17038.958,E2 -17038.958} C_VEL
LIN {X 0,Y 293.159,Z 879.276,A -85,B 0,C 180,E1 -17040.719,E2 -17040.719} C_VEL
LIN {X 0,Y 292.016,Z 871.599,A -85,B 0,C 180,E1 -17041.973,E2 -17041.973} C_VEL
LIN {X 0,Y 291.354,Z 867.005,A -85,B 0,C 180,E1 -17042.728,E2 -17042.728} C_VEL
LIN {X 0,Y 290.413,Z 862.46,A -85,B 0,C 180,E1 -17043.552,E2 -17043.552} C_VEL
LIN {X 0,Y 289.953,Z 859.009,A -85,B 0,C 180,E1 -17044.135,E2 -17044.135} C_VEL
LIN {X 0,Y 288.493,Z 852.208,A -85,B 0,C 180,E1 -17045.541,E2 -17045.541} C_VEL
LIN {X 0,Y 288.38,Z 849.725,A -85,B 0,C 180,E1 -17045.986,E2 -17045.986} C_VEL
LIN {X 0,Y 289.313,Z 844.596,A -85,B 0,C 180,E1 -17048.178,E2 -17048.178} C_VEL
LIN {X 0,Y 288.91,Z 840.43,A -85,B 0,C 180,E1 -17050.073,E2 -17050.073} C_VEL
LIN {X 0,Y 287.703,Z 834.07,A -85,B 0,C 180,E1 -17053.158,E2 -17053.158} C_VEL
LIN {X 0,Y 286.543,Z 827.971,A -85,B 0,C 180,E1 -17056.273,E2 -17056.273} C_VEL
LIN {X 0,Y 286.815,Z 825.521,A -85,B 0,C 180,E1 -17059.433,E2 -17059.433} C_VEL
LIN {X 0,Y 287.022,Z 824.952,A -85,B 0,C 180,E1 -17060.459,E2 -17060.459} C_VEL
LIN {X 0,Y 286.967,Z 824.53,A -85,B 0,C 180,E1 -17062.689,E2 -17062.689} C_VEL
LIN {X 0,Y 290.266,Z 827.321,A -85,B 0,C 180,E1 -17065.411,E2 -17065.411} C_VEL
LIN {X 0,Y 294.805,Z 832.41,A -85,B 0,C 180,E1 -17068.368,E2 -17068.368} C_VEL
LIN {X 0,Y 298.893,Z 840.652,A -85,B 0,C 180,E1 -17071.248,E2 -17071.248} C_VEL
LIN {X 0,Y 301.501,Z 847.289,A -85,B 0,C 180,E1 -17073.213,E2 -17073.213} C_VEL
LIN {X 0,Y 303.803,Z 855.309,A -85,B 0,C 180,E1 -17075.392,E2 -17075.392} C_VEL
LIN {X 0,Y 304.649,Z 859.753,A -85,B 0,C 180,E1 -17076.512,E2 -17076.512} C_VEL
LIN {X 0,Y 302.167,Z 868.834,A -85,B 0,C 180,E1 -17078.152,E2 -17078.152} C_VEL
LIN {X 0,Y 299.326,Z 877.829,A -85,B 0,C 180,E1 -17080.096,E2 -17080.096} C_VEL
LIN {X 0,Y 296.243,Z 886.16,A -85,B 0,C 180,E1 -17082.394,E2 -17082.394} C_VEL
LIN {X 0,Y 293.67,Z 892.594,A -85,B 0,C 180,E1 -17084.737,E2 -17084.737} C_VEL
LIN {X 0,Y 291.609,Z 896.964,A -85,B 0,C 180,E1 -17086.764,E2 -17086.764} C_VEL
LIN {X 0,Y 289.857,Z 900.189,A -85,B 0,C 180,E1 -17088.815,E2 -17088.815} C_VEL
LIN {X 0,Y 288.811,Z 901.893,A -85,B 0,C 180,E1 -17090.192,E2 -17090.192} C_VEL
LIN {X 0,Y 287.182,Z 903.849,A -85,B 0,C 180,E1 -17092.972,E2 -17092.972} C_VEL
LIN {X 0,Y 286.581,Z 904.282,A -85,B 0,C 180,E1 -17094.371,E2 -17094.371} C_VEL
LIN {X 0,Y 286.083,Z 904.299,A -85,B 0,C 180,E1 -17095.774,E2 -17095.774} C_VEL
LIN {X 0,Y 285.21,Z 903.084,A -85,B 0,C 180,E1 -17098.588,E2 -17098.588} C_VEL
LIN {X 0,Y 284.769,Z 901.815,A -85,B 0,C 180,E1 -17100,E2 -17100} C_VEL
LIN {X 0,Y 284.661,Z 899.19,A -85,B 0,C 180,E1 -17102.122,E2 -17102.122} C_VEL
LIN {X 0,Y 284.411,Z 895.613,A -85,B 0,C 180,E1 -17104.251,E2 -17104.251} C_VEL
LIN {X 0,Y 284.888,Z 890.929,A -85,B 0,C 180,E1 -17106.374,E2 -17106.374} C_VEL
LIN {X 0,Y 285.2,Z 886.15,A -85,B 0,C 180,E1 -17108.146,E2 -17108.146} C_VEL
LIN {X 0,Y 285.575,Z 880.461,A -85,B 0,C 180,E1 -17109.92,E2 -17109.92} C_VEL
LIN {X 0,Y 286.135,Z 873.814,A -85,B 0,C 180,E1 -17111.691,E2 -17111.691} C_VEL
LIN {X 0,Y 286.84,Z 865.71,A -85,B 0,C 180,E1 -17113.46,E2 -17113.46} C_VEL
LIN {X 0,Y 287.547,Z 857.185,A -85,B 0,C 180,E1 -17115.052,E2 -17115.052} C_VEL
LIN {X 0,Y 288.321,Z 848.27,A -85,B 0,C 180,E1 -17116.461,E2 -17116.461} C_VEL
LIN {X 0,Y 289.164,Z 837.655,A -85,B 0,C 180,E1 -17117.882,E2 -17117.882} C_VEL
LIN {X 0,Y 288.68,Z 834.461,A -85,B 0,C 180,E1 -17118.287,E2 -17118.287} C_VEL
LIN {X 0,Y 285.831,Z 823.087,A -85,B 0,C 180,E1 -17119.59,E2 -17119.59} C_VEL
LIN {X 0,Y 284.365,Z 817.055,A -85,B 0,C 180,E1 -17120.197,E2 -17120.197} C_VEL
LIN {X 0,Y 284.3,Z 817.072,A -85,B 0,C 180,E1 -17123.839,E2 -17123.839} C_VEL
LIN {X 0,Y 284.293,Z 817.06,A -85,B 0,C 180,E1 -17127.129,E2 -17127.129} C_VEL
LIN {X 0,Y 284.281,Z 817.071,A -85,B 0,C 180,E1 -17130.083,E2 -17130.083} C_VEL
LIN {X 0,Y 284.312,Z 817.055,A -85,B 0,C 180,E1 -17132.945,E2 -17132.945} C_VEL
LIN {X 0,Y 284.325,Z 817.062,A -85,B 0,C 180,E1 -17136.387,E2 -17136.387} C_VEL
LIN {X 0,Y 284.289,Z 817.073,A -85,B 0,C 180,E1 -17139.998,E2 -17139.998} C_VEL
LIN {X 0,Y 284.242,Z 817.08,A -85,B 0,C 180,E1 -17144.187,E2 -17144.187} C_VEL
LIN {X 0,Y 284.247,Z 817.08,A -85,B 0,C 180,E1 -17148.117,E2 -17148.117} C_VEL
LIN {X 0,Y 284.308,Z 817.068,A -85,B 0,C 180,E1 -17152.282,E2 -17152.282} C_VEL
LIN {X 0,Y 284.314,Z 817.068,A -85,B 0,C 180,E1 -17155.349,E2 -17155.349} C_VEL
LIN {X 0,Y 284.301,Z 817.064,A -85,B 0,C 180,E1 -17158.724,E2 -17158.724} C_VEL
LIN {X 0,Y 284.402,Z 817.05,A -85,B 0,C 180,E1 -17162.825,E2 -17162.825} C_VEL
LIN {X 0,Y 284.439,Z 817.154,A -85,B 0,C 180,E1 -17165.063,E2 -17165.063} C_VEL
LIN {X 0,Y 285.811,Z 820.958,A -85,B 0,C 180,E1 -17165.481,E2 -17165.481} C_VEL
LIN {X 0,Y 289.679,Z 830.858,A -85,B 0,C 180,E1 -17166.736,E2 -17166.736} C_VEL
LIN {X 0,Y 293.028,Z 841.399,A -85,B 0,C 180,E1 -17168.237,E2 -17168.237} C_VEL
LIN {X 0,Y 294.69,Z 847.552,A -85,B 0,C 180,E1 -17169.213,E2 -17169.213} C_VEL
LIN {X 0,Y 293.267,Z 858.123,A -85,B 0,C 180,E1 -17170.759,E2 -17170.759} C_VEL
LIN {X 0,Y 291.853,Z 867.567,A -85,B 0,C 180,E1 -17172.48,E2 -17172.48} C_VEL
LIN {X 0,Y 290.312,Z 875.331,A -85,B 0,C 180,E1 -17174.194,E2 -17174.194} C_VEL
LIN {X 0,Y 288.906,Z 882.878,A -85,B 0,C 180,E1 -17176.278,E2 -17176.278} C_VEL
LIN {X 0,Y 287.731,Z 889.757,A -85,B 0,C 180,E1 -17178.729,E2 -17178.729} C_VEL
LIN {X 0,Y 286.517,Z 894.394,A -85,B 0,C 180,E1 -17180.823,E2 -17180.823} C_VEL
LIN {X 0,Y 285.701,Z 897.916,A -85,B 0,C 180,E1 -17182.933,E2 -17182.933} C_VEL
LIN {X 0,Y 285.306,Z 899.732,A -85,B 0,C 180,E1 -17184.343,E2 -17184.343} C_VEL
LIN {X 0,Y 285.25,Z 901.062,A -85,B 0,C 180,E1 -17185.759,E2 -17185.759} C_VEL
LIN {X 0,Y 284.842,Z 902.641,A -85,B 0,C 180,E1 -17188.584,E2 -17188.584} C_VEL
LIN {X 0,Y 284.783,Z 902.871,A -85,B 0,C 180,E1 -17189.997,E2 -17189.997} C_VEL
LIN {X 0,Y 285.023,Z 902.102,A -85,B 0,C 180,E1 -17192.824,E2 -17192.824} C_VEL
LIN {X 0,Y 285.231,Z 901.159,A -85,B 0,C 180,E1 -17194.237,E2 -17194.237} C_VEL
LIN {X 0,Y 285.292,Z 899.869,A -85,B 0,C 180,E1 -17195.652,E2 -17195.652} C_VEL
LIN {X 0,Y 285.916,Z 897.062,A -85,B 0,C 180,E1 -17197.767,E2 -17197.767} C_VEL
LIN {X 0,Y 286.982,Z 893.218,A -85,B 0,C 180,E1 -17199.868,E2 -17199.868} C_VEL
LIN {X 0,Y 288.008,Z 888.306,A -85,B 0,C 180,E1 -17201.968,E2 -17201.968} C_VEL
LIN {X 0,Y 289.098,Z 882.131,A -85,B 0,C 180,E1 -17204.067,E2 -17204.067} C_VEL
LIN {X 0,Y 290.609,Z 874.357,A -85,B 0,C 180,E1 -17206.145,E2 -17206.145} C_VEL
LIN {X 0,Y 291.993,Z 866.427,A -85,B 0,C 180,E1 -17207.868,E2 -17207.868} C_VEL
LIN {X 0,Y 293.535,Z 856.729,A -85,B 0,C 180,E1 -17209.582,E2 -17209.582} C_VEL
LIN {X 0,Y 294.632,Z 849.007,A -85,B 0,C 180,E1 -17210.697,E2 -17210.697} C_VEL
LIN {X 0,Y 294.627,Z 847.204,A -85,B 0,C 180,E1 -17210.963,E2 -17210.963} C_VEL
LIN {X 0,Y 291.88,Z 837.352,A -85,B 0,C 180,E1 -17212.48,E2 -17212.48} C_VEL
LIN {X 0,Y 288.063,Z 826.577,A -85,B 0,C 180,E1 -17213.947,E2 -17213.947} C_VEL
LIN {X 0,Y 284.453,Z 817.322,A -85,B 0,C 180,E1 -17215.046,E2 -17215.046} C_VEL
LIN {X 0,Y 284.419,Z 817.057,A -85,B 0,C 180,E1 -17215.08,E2 -17215.08} C_VEL
LIN {X 0,Y 284.327,Z 817.069,A -85,B 0,C 180,E1 -17218.008,E2 -17218.008} C_VEL
LIN {X 0,Y 284.29,Z 817.073,A -85,B 0,C 180,E1 -17221.271,E2 -17221.271} C_VEL
LIN {X 0,Y 284.355,Z 817.065,A -85,B 0,C 180,E1 -17225.351,E2 -17225.351} C_VEL
LIN {X 0,Y 284.33,Z 817.07,A -85,B 0,C 180,E1 -17228.162,E2 -17228.162} C_VEL
LIN {X 0,Y 284.346,Z 817.069,A -85,B 0,C 180,E1 -17232.141,E2 -17232.141} C_VEL
LIN {X 0,Y 284.344,Z 817.066,A -85,B 0,C 180,E1 -17236.206,E2 -17236.206} C_VEL
LIN {X 0,Y 284.356,Z 817.065,A -85,B 0,C 180,E1 -17240.013,E2 -17240.013} C_VEL
LIN {X 0,Y 284.344,Z 817.064,A -85,B 0,C 180,E1 -17243.616,E2 -17243.616} C_VEL
LIN {X 0,Y 284.295,Z 817.071,A -85,B 0,C 180,E1 -17247.188,E2 -17247.188} C_VEL
LIN {X 0,Y 284.346,Z 817.059,A -85,B 0,C 180,E1 -17250.374,E2 -17250.374} C_VEL
LIN {X 0,Y 284.364,Z 817.058,A -85,B 0,C 180,E1 -17253.585,E2 -17253.585} C_VEL
LIN {X 0,Y 284.352,Z 817.065,A -85,B 0,C 180,E1 -17256.706,E2 -17256.706} C_VEL
LIN {X 0,Y 284.389,Z 817.062,A -85,B 0,C 180,E1 -17261.26,E2 -17261.26} C_VEL
LIN {X 0,Y 284.477,Z 817.039,A -85,B 0,C 180,E1 -17264.458,E2 -17264.458} C_VEL
LIN {X 0,Y 284.475,Z 817.051,A -85,B 0,C 180,E1 -17268.601,E2 -17268.601} C_VEL
LIN {X 0,Y 284.641,Z 817.023,A -85,B 0,C 180,E1 -17271.48,E2 -17271.48} C_VEL
LIN {X 0,Y 284.582,Z 817.039,A -85,B 0,C 180,E1 -17274.331,E2 -17274.331} C_VEL
LIN {X 0,Y 284.84,Z 817.005,A -85,B 0,C 180,E1 -17278.586,E2 -17278.586} C_VEL
LIN {X 0,Y 284.839,Z 817.008,A -85,B 0,C 180,E1 -17281.414,E2 -17281.414} C_VEL
LIN {X 0,Y 284.726,Z 817.021,A -85,B 0,C 180,E1 -17282.775,E2 -17282.775} C_VEL
LIN {X 0,Y 284.03,Z 817.112,A -85,B 0,C 180,E1 -17283.954,E2 -17283.954} C_VEL
LIN {X 0,Y 281.12,Z 817.472,A -85,B 0,C 180,E1 -17285.874,E2 -17285.874} C_VEL
LIN {X 0,Y 278.683,Z 817.772,A -85,B 0,C 180,E1 -17287.434,E2 -17287.434} C_VEL
LIN {X 0,Y 277.671,Z 817.895,A -85,B 0,C 180,E1 -17288.643,E2 -17288.643} C_VEL
LIN {X 0,Y 277.607,Z 817.904,A -85,B 0,C 180,E1 -17289.053,E2 -17289.053} C_VEL
LIN {X 0,Y 277.402,Z 817.924,A -85,B 0,C 180,E1 -17293.18,E2 -17293.18} C_VEL
LIN {X 0,Y 277.39,Z 817.934,A -85,B 0,C 180,E1 -17296.183,E2 -17296.183} C_VEL
LIN {X 0,Y 277.329,Z 817.943,A -85,B 0,C 180,E1 -17300.35,E2 -17300.35} C_VEL
LIN {X 0,Y 277.262,Z 817.95,A -85,B 0,C 180,E1 -17304.152,E2 -17304.152} C_VEL
LIN {X 0,Y 277.255,Z 817.944,A -85,B 0,C 180,E1 -17307.484,E2 -17307.484} C_VEL
LIN {X 0,Y 277.234,Z 817.949,A -85,B 0,C 180,E1 -17310.474,E2 -17310.474} C_VEL
LIN {X 0,Y 277.232,Z 817.954,A -85,B 0,C 180,E1 -17313.898,E2 -17313.898} C_VEL
LIN {X 0,Y 277.298,Z 818.053,A -85,B 0,C 180,E1 -17317.012,E2 -17317.012} C_VEL
LIN {X 0,Y 279.025,Z 826.363,A -85,B 0,C 180,E1 -17321.873,E2 -17321.873} C_VEL
LIN {X 0,Y 280.336,Z 832.986,A -85,B 0,C 180,E1 -17325.42,E2 -17325.42} C_VEL
LIN {X 0,Y 281.689,Z 840.169,A -85,B 0,C 180,E1 -17329.047,E2 -17329.047} C_VEL
LIN {X 0,Y 282.336,Z 844.305,A -85,B 0,C 180,E1 -17331.036,E2 -17331.036} C_VEL
LIN {X 0,Y 281.744,Z 848.608,A -85,B 0,C 180,E1 -17332.961,E2 -17332.961} C_VEL
LIN {X 0,Y 280.317,Z 856.783,A -85,B 0,C 180,E1 -17336.529,E2 -17336.529} C_VEL
LIN {X 0,Y 278.631,Z 867.96,A -85,B 0,C 180,E1 -17341.367,E2 -17341.367} C_VEL
LIN {X 0,Y 278.014,Z 872.823,A -85,B 0,C 180,E1 -17343.435,E2 -17343.435} C_VEL
LIN {X 0,Y 280.283,Z 886.894,A -85,B 0,C 180,E1 -17344.268,E2 -17344.268} C_VEL
LIN {X 0,Y 281.766,Z 900.131,A -85,B 0,C 180,E1 -17345.298,E2 -17345.298} C_VEL
LIN {X 0,Y 282.375,Z 912.875,A -85,B 0,C 180,E1 -17346.536,E2 -17346.536} C_VEL
LIN {X 0,Y 282.271,Z 923.95,A -85,B 0,C 180,E1 -17347.844,E2 -17347.844} C_VEL
LIN {X 0,Y 281.748,Z 934.641,A -85,B 0,C 180,E1 -17349.373,E2 -17349.373} C_VEL
LIN {X 0,Y 281.545,Z 940.229,A -85,B 0,C 180,E1 -17350.309,E2 -17350.309} C_VEL
LIN {X 0,Y 279.831,Z 949.548,A -85,B 0,C 180,E1 -17352.085,E2 -17352.085} C_VEL
LIN {X 0,Y 278.111,Z 958.658,A -85,B 0,C 180,E1 -17354.24,E2 -17354.24} C_VEL
LIN {X 0,Y 277.167,Z 966.087,A -85,B 0,C 180,E1 -17356.438,E2 -17356.438} C_VEL
LIN {X 0,Y 276.447,Z 972.891,A -85,B 0,C 180,E1 -17359.011,E2 -17359.011} C_VEL
LIN {X 0,Y 276.245,Z 977.445,A -85,B 0,C 180,E1 -17361.222,E2 -17361.222} C_VEL
LIN {X 0,Y 276.263,Z 980.059,A -85,B 0,C 180,E1 -17362.813,E2 -17362.813} C_VEL
LIN {X 0,Y 276.375,Z 981.862,A -85,B 0,C 180,E1 -17364.165,E2 -17364.165} C_VEL
LIN {X 0,Y 276.631,Z 983.377,A -85,B 0,C 180,E1 -17365.632,E2 -17365.632} C_VEL
LIN {X 0,Y 276.757,Z 984.447,A -85,B 0,C 180,E1 -17367.091,E2 -17367.091} C_VEL
LIN {X 0,Y 276.891,Z 985.107,A -85,B 0,C 180,E1 -17368.548,E2 -17368.548} C_VEL
LIN {X 0,Y 277.024,Z 985.351,A -85,B 0,C 180,E1 -17370.003,E2 -17370.003} C_VEL
LIN {X 0,Y 276.892,Z 985.098,A -85,B 0,C 180,E1 -17371.457,E2 -17371.457} C_VEL
LIN {X 0,Y 276.759,Z 984.432,A -85,B 0,C 180,E1 -17372.914,E2 -17372.914} C_VEL
LIN {X 0,Y 276.656,Z 983.358,A -85,B 0,C 180,E1 -17374.373,E2 -17374.373} C_VEL
LIN {X 0,Y 276.406,Z 981.835,A -85,B 0,C 180,E1 -17375.84,E2 -17375.84} C_VEL
LIN {X 0,Y 276.274,Z 978.704,A -85,B 0,C 180,E1 -17378.045,E2 -17378.045} C_VEL
LIN {X 0,Y 276.789,Z 970.527,A -85,B 0,C 180,E1 -17382.466,E2 -17382.466} C_VEL
LIN {X 0,Y 277.658,Z 965.359,A -85,B 0,C 180,E1 -17384.665,E2 -17384.665} C_VEL
LIN {X 0,Y 279.678,Z 956.738,A -85,B 0,C 180,E1 -17387.553,E2 -17387.553} C_VEL
LIN {X 0,Y 281.788,Z 948.832,A -85,B 0,C 180,E1 -17389.678,E2 -17389.678} C_VEL
LIN {X 0,Y 283.743,Z 941.256,A -85,B 0,C 180,E1 -17391.431,E2 -17391.431} C_VEL
LIN {X 0,Y 285.587,Z 930.704,A -85,B 0,C 180,E1 -17393.566,E2 -17393.566} C_VEL
LIN {X 0,Y 287.482,Z 920.427,A -85,B 0,C 180,E1 -17395.349,E2 -17395.349} C_VEL
LIN {X 0,Y 288.497,Z 912.77,A -85,B 0,C 180,E1 -17396.594,E2 -17396.594} C_VEL
LIN {X 0,Y 288.919,Z 900.018,A -85,B 0,C 180,E1 -17398.632,E2 -17398.632} C_VEL
LIN {X 0,Y 288.458,Z 886.66,A -85,B 0,C 180,E1 -17400.776,E2 -17400.776} C_VEL
LIN {X 0,Y 287.506,Z 876.373,A -85,B 0,C 180,E1 -17402.535,E2 -17402.535} C_VEL
LIN {X 0,Y 286.809,Z 870.553,A -85,B 0,C 180,E1 -17403.577,E2 -17403.577} C_VEL
LIN {X 0,Y 285.707,Z 862.544,A -85,B 0,C 180,E1 -17405.124,E2 -17405.124} C_VEL
LIN {X 0,Y 284.818,Z 856.912,A -85,B 0,C 180,E1 -17406.316,E2 -17406.316} C_VEL
LIN {X 0,Y 284.75,Z 855.065,A -85,B 0,C 180,E1 -17406.643,E2 -17406.643} C_VEL
LIN {X 0,Y 282.808,Z 845.137,A -85,B 0,C 180,E1 -17409.401,E2 -17409.401} C_VEL
LIN {X 0,Y 281.656,Z 839.706,A -85,B 0,C 180,E1 -17411.533,E2 -17411.533} C_VEL
LIN {X 0,Y 280.993,Z 836.122,A -85,B 0,C 180,E1 -17413.504,E2 -17413.504} C_VEL
LIN {X 0,Y 281.007,Z 832.267,A -85,B 0,C 180,E1 -17416.496,E2 -17416.496} C_VEL
LIN {X 0,Y 281.588,Z 831.125,A -85,B 0,C 180,E1 -17418.485,E2 -17418.485} C_VEL
LIN {X 0,Y 282.732,Z 830.677,A -85,B 0,C 180,E1 -17420.409,E2 -17420.409} C_VEL
LIN {X 0,Y 284.326,Z 831.07,A -85,B 0,C 180,E1 -17422.28,E2 -17422.28} C_VEL
LIN {X 0,Y 287.152,Z 833.596,A -85,B 0,C 180,E1 -17425.015,E2 -17425.015} C_VEL
LIN {X 0,Y 290.997,Z 838.034,A -85,B 0,C 180,E1 -17427.904,E2 -17427.904} C_VEL
LIN {X 0,Y 294.872,Z 846.735,A -85,B 0,C 180,E1 -17431.117,E2 -17431.117} C_VEL
LIN {X 0,Y 297.171,Z 853.732,A -85,B 0,C 180,E1 -17433.298,E2 -17433.298} C_VEL
LIN {X 0,Y 298.698,Z 860.575,A -85,B 0,C 180,E1 -17435.261,E2 -17435.261} C_VEL
LIN {X 0,Y 298.995,Z 862.776,A -85,B 0,C 180,E1 -17435.869,E2 -17435.869} C_VEL
LIN {X 0,Y 298.358,Z 865.466,A -85,B 0,C 180,E1 -17436.394,E2 -17436.394} C_VEL
LIN {X 0,Y 296.156,Z 872.217,A -85,B 0,C 180,E1 -17437.685,E2 -17437.685} C_VEL
LIN {X 0,Y 293.642,Z 879.512,A -85,B 0,C 180,E1 -17439.328,E2 -17439.328} C_VEL
LIN {X 0,Y 290.335,Z 887.729,A -85,B 0,C 180,E1 -17441.658,E2 -17441.658} C_VEL
LIN {X 0,Y 287.908,Z 893.324,A -85,B 0,C 180,E1 -17443.697,E2 -17443.697} C_VEL
